REGION Network 8: MATERIAL ADDITION PROCESS SELECT
   RUNG wire#powerrail
      { S7_Templates := "SrcType := Int" } EQ_Contact(in1 := "MODE SELECTION DB"."MODE BUFF", in2 := 1)
      { S7_Templates := "SrcType := Int" } EQ_Contact(in1 := "MFG PROCESS_DB"."AUTO BUFF", in2 := 60)
      Coil( "AUTO ALARM DB"."MFG PROCESS"."MATERIAL ADDITION PROCESS SELECT" )
   END_RUNG
   // the same network as SCL:
   "AUTO ALARM DB"."MFG PROCESS"."MATERIAL ADDITION PROCESS SELECT" := ("MODE SELECTION DB"."MODE BUFF" = 1) AND ("MFG PROCESS_DB"."AUTO BUFF" = 60);
END_REGION

REGION Network 9: MATERIAL ADDITION MATERIAL ADDED TEXT
   RUNG wire#powerrail
      { S7_Templates := "SrcType := Int" } EQ_Contact(in1 := "MODE SELECTION DB"."MODE BUFF", in2 := 1)
      { S7_Templates := "SrcType := Int" } EQ_Contact(in1 := "MFG PROCESS_DB"."AUTO BUFF", in2 := 65)
      Coil( "AUTO ALARM DB"."MFG PROCESS"."MATERIAL ADDITION MATERIAL ADDED TEXT" )
   END_RUNG
   // the same network as SCL:
   "AUTO ALARM DB"."MFG PROCESS"."MATERIAL ADDITION MATERIAL ADDED TEXT" := ("MODE SELECTION DB"."MODE BUFF" = 1) AND ("MFG PROCESS_DB"."AUTO BUFF" = 65);
END_REGION

REGION Network 10: MATERIAL ADDITION DO YOU WANT TO ADD SORBITOL SELECT
   RUNG wire#powerrail
      { S7_Templates := "SrcType := Int" } EQ_Contact(in1 := "MODE SELECTION DB"."MODE BUFF", in2 := 1)
      { S7_Templates := "SrcType := Int" } EQ_Contact(in1 := "MFG PROCESS_DB"."AUTO BUFF", in2 := 75)
      Coil( "AUTO ALARM DB"."MFG PROCESS"."MATERIAL ADDITION DO YOU WANT TO ADD SORBITOL SELECT" )
   END_RUNG
   // the same network as SCL:
   "AUTO ALARM DB"."MFG PROCESS"."MATERIAL ADDITION DO YOU WANT TO ADD SORBITOL SELECT" := ("MODE SELECTION DB"."MODE BUFF" = 1) AND ("MFG PROCESS_DB"."AUTO BUFF" = 75);
END_REGION

REGION Network 11: MATERIAL ADDITION OF SORBITOL OVER
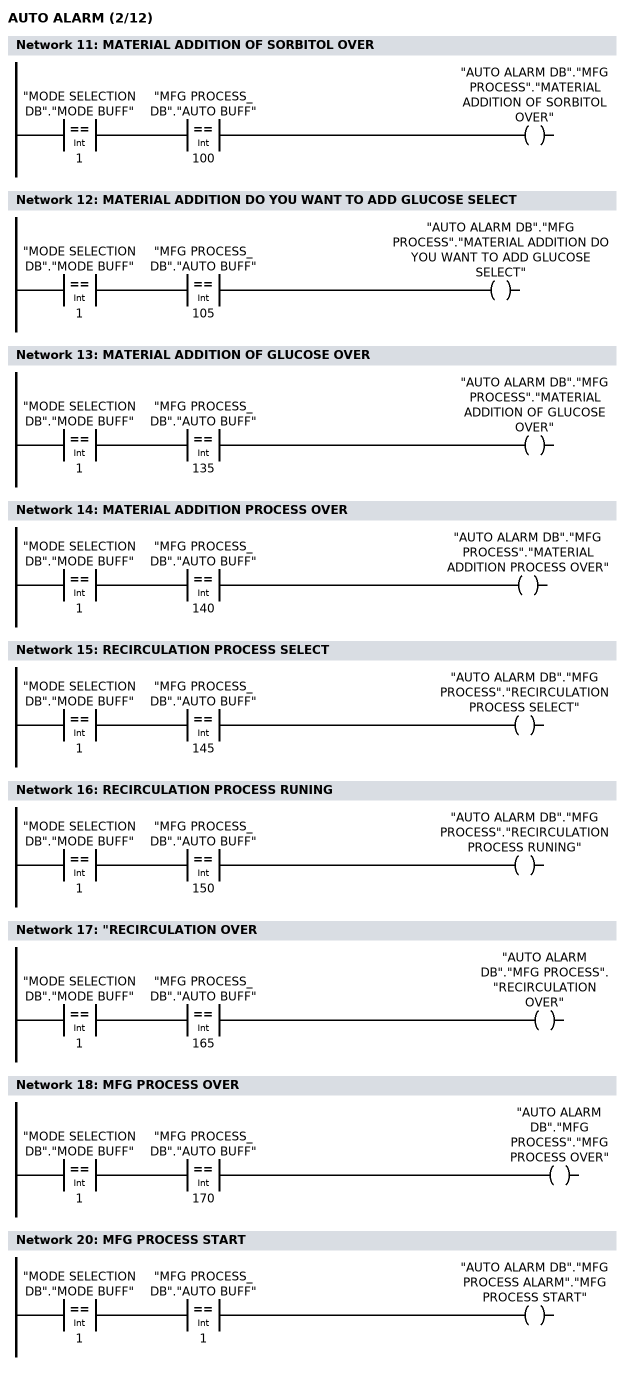
   RUNG wire#powerrail
      { S7_Templates := "SrcType := Int" } EQ_Contact(in1 := "MODE SELECTION DB"."MODE BUFF", in2 := 1)
      { S7_Templates := "SrcType := Int" } EQ_Contact(in1 := "MFG PROCESS_DB"."AUTO BUFF", in2 := 100)
      Coil( "AUTO ALARM DB"."MFG PROCESS"."MATERIAL ADDITION OF SORBITOL OVER" )
   END_RUNG
   // the same network as SCL:
   "AUTO ALARM DB"."MFG PROCESS"."MATERIAL ADDITION OF SORBITOL OVER" := ("MODE SELECTION DB"."MODE BUFF" = 1) AND ("MFG PROCESS_DB"."AUTO BUFF" = 100);
END_REGION

REGION Network 12: MATERIAL ADDITION DO YOU WANT TO ADD GLUCOSE SELECT
   RUNG wire#powerrail
      { S7_Templates := "SrcType := Int" } EQ_Contact(in1 := "MODE SELECTION DB"."MODE BUFF", in2 := 1)
      { S7_Templates := "SrcType := Int" } EQ_Contact(in1 := "MFG PROCESS_DB"."AUTO BUFF", in2 := 105)
      Coil( "AUTO ALARM DB"."MFG PROCESS"."MATERIAL ADDITION DO YOU WANT TO ADD GLUCOSE SELECT" )
   END_RUNG
   // the same network as SCL:
   "AUTO ALARM DB"."MFG PROCESS"."MATERIAL ADDITION DO YOU WANT TO ADD GLUCOSE SELECT" := ("MODE SELECTION DB"."MODE BUFF" = 1) AND ("MFG PROCESS_DB"."AUTO BUFF" = 105);
END_REGION

REGION Network 13: MATERIAL ADDITION OF GLUCOSE OVER
   RUNG wire#powerrail
      { S7_Templates := "SrcType := Int" } EQ_Contact(in1 := "MODE SELECTION DB"."MODE BUFF", in2 := 1)
      { S7_Templates := "SrcType := Int" } EQ_Contact(in1 := "MFG PROCESS_DB"."AUTO BUFF", in2 := 135)
      Coil( "AUTO ALARM DB"."MFG PROCESS"."MATERIAL ADDITION OF GLUCOSE OVER" )
   END_RUNG
   // the same network as SCL:
   "AUTO ALARM DB"."MFG PROCESS"."MATERIAL ADDITION OF GLUCOSE OVER" := ("MODE SELECTION DB"."MODE BUFF" = 1) AND ("MFG PROCESS_DB"."AUTO BUFF" = 135);
END_REGION

REGION Network 14: MATERIAL ADDITION PROCESS OVER
   RUNG wire#powerrail
      { S7_Templates := "SrcType := Int" } EQ_Contact(in1 := "MODE SELECTION DB"."MODE BUFF", in2 := 1)
      { S7_Templates := "SrcType := Int" } EQ_Contact(in1 := "MFG PROCESS_DB"."AUTO BUFF", in2 := 140)
      Coil( "AUTO ALARM DB"."MFG PROCESS"."MATERIAL ADDITION PROCESS OVER" )
   END_RUNG
   // the same network as SCL:
   "AUTO ALARM DB"."MFG PROCESS"."MATERIAL ADDITION PROCESS OVER" := ("MODE SELECTION DB"."MODE BUFF" = 1) AND ("MFG PROCESS_DB"."AUTO BUFF" = 140);
END_REGION

REGION Network 15: RECIRCULATION PROCESS SELECT
   RUNG wire#powerrail
      { S7_Templates := "SrcType := Int" } EQ_Contact(in1 := "MODE SELECTION DB"."MODE BUFF", in2 := 1)
      { S7_Templates := "SrcType := Int" } EQ_Contact(in1 := "MFG PROCESS_DB"."AUTO BUFF", in2 := 145)
      Coil( "AUTO ALARM DB"."MFG PROCESS"."RECIRCULATION PROCESS SELECT" )
   END_RUNG
   // the same network as SCL:
   "AUTO ALARM DB"."MFG PROCESS"."RECIRCULATION PROCESS SELECT" := ("MODE SELECTION DB"."MODE BUFF" = 1) AND ("MFG PROCESS_DB"."AUTO BUFF" = 145);
END_REGION

REGION Network 16: RECIRCULATION PROCESS RUNING
   RUNG wire#powerrail
      { S7_Templates := "SrcType := Int" } EQ_Contact(in1 := "MODE SELECTION DB"."MODE BUFF", in2 := 1)
      { S7_Templates := "SrcType := Int" } EQ_Contact(in1 := "MFG PROCESS_DB"."AUTO BUFF", in2 := 150)
      Coil( "AUTO ALARM DB"."MFG PROCESS"."RECIRCULATION PROCESS RUNING" )
   END_RUNG
   // the same network as SCL:
   "AUTO ALARM DB"."MFG PROCESS"."RECIRCULATION PROCESS RUNING" := ("MODE SELECTION DB"."MODE BUFF" = 1) AND ("MFG PROCESS_DB"."AUTO BUFF" = 150);
END_REGION

REGION Network 17: "RECIRCULATION OVER
   RUNG wire#powerrail
      { S7_Templates := "SrcType := Int" } EQ_Contact(in1 := "MODE SELECTION DB"."MODE BUFF", in2 := 1)
      { S7_Templates := "SrcType := Int" } EQ_Contact(in1 := "MFG PROCESS_DB"."AUTO BUFF", in2 := 165)
      Coil( "AUTO ALARM DB"."MFG PROCESS"."RECIRCULATION OVER" )
   END_RUNG
   // the same network as SCL:
   "AUTO ALARM DB"."MFG PROCESS"."RECIRCULATION OVER" := ("MODE SELECTION DB"."MODE BUFF" = 1) AND ("MFG PROCESS_DB"."AUTO BUFF" = 165);
END_REGION

REGION Network 18: MFG PROCESS OVER
   RUNG wire#powerrail
      { S7_Templates := "SrcType := Int" } EQ_Contact(in1 := "MODE SELECTION DB"."MODE BUFF", in2 := 1)
      { S7_Templates := "SrcType := Int" } EQ_Contact(in1 := "MFG PROCESS_DB"."AUTO BUFF", in2 := 170)
      Coil( "AUTO ALARM DB"."MFG PROCESS"."MFG PROCESS OVER" )
   END_RUNG
   // the same network as SCL:
   "AUTO ALARM DB"."MFG PROCESS"."MFG PROCESS OVER" := ("MODE SELECTION DB"."MODE BUFF" = 1) AND ("MFG PROCESS_DB"."AUTO BUFF" = 170);
END_REGION

REGION Network 19: ///////////////////////////////MFG ALARM /////////////////////////////////////
END_REGION

REGION Network 20: MFG PROCESS START
   RUNG wire#powerrail
      { S7_Templates := "SrcType := Int" } EQ_Contact(in1 := "MODE SELECTION DB"."MODE BUFF", in2 := 1)
      { S7_Templates := "SrcType := Int" } EQ_Contact(in1 := "MFG PROCESS_DB"."AUTO BUFF", in2 := 1)
      Coil( "AUTO ALARM DB"."MFG PROCESS ALARM"."MFG PROCESS START" )
   END_RUNG
   // the same network as SCL:
   "AUTO ALARM DB"."MFG PROCESS ALARM"."MFG PROCESS START" := ("MODE SELECTION DB"."MODE BUFF" = 1) AND ("MFG PROCESS_DB"."AUTO BUFF" = 1);
END_REGION

REGION Network 21: PURIFIED WATER PROCESS START
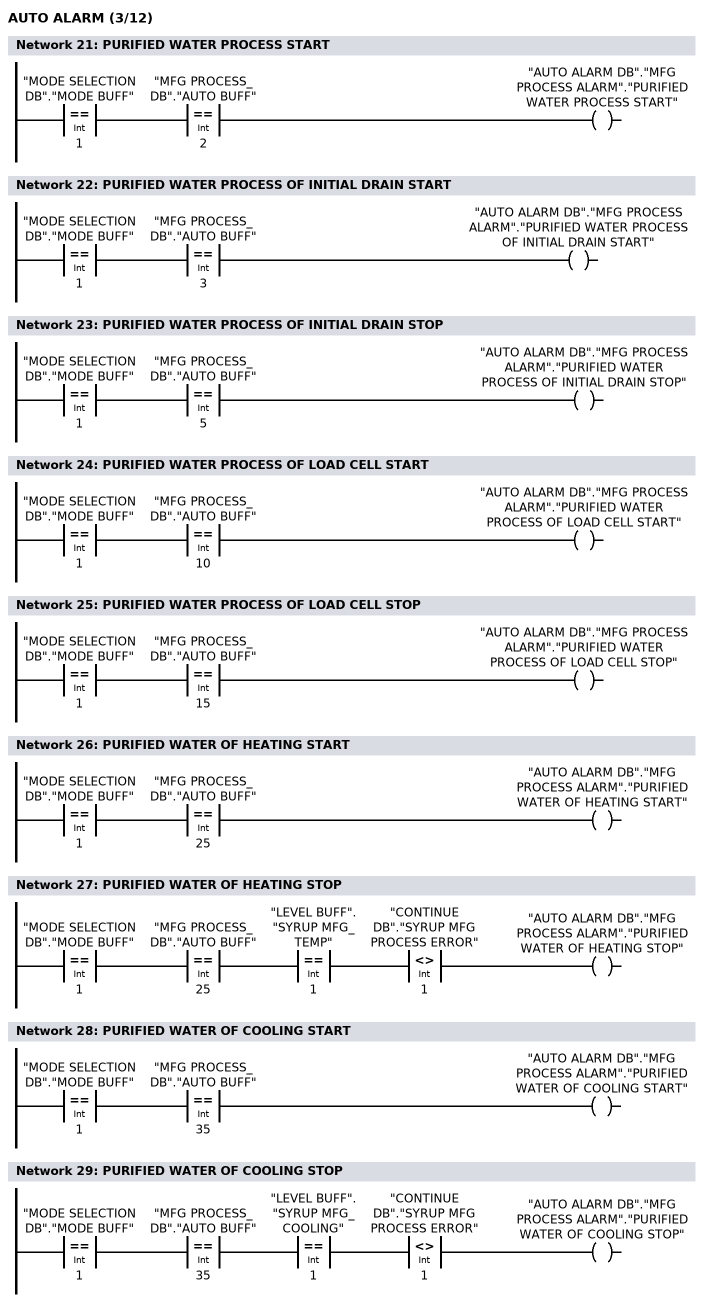
   RUNG wire#powerrail
      { S7_Templates := "SrcType := Int" } EQ_Contact(in1 := "MODE SELECTION DB"."MODE BUFF", in2 := 1)
      { S7_Templates := "SrcType := Int" } EQ_Contact(in1 := "MFG PROCESS_DB"."AUTO BUFF", in2 := 2)
      Coil( "AUTO ALARM DB"."MFG PROCESS ALARM"."PURIFIED WATER PROCESS START" )
   END_RUNG
   // the same network as SCL:
   "AUTO ALARM DB"."MFG PROCESS ALARM"."PURIFIED WATER PROCESS START" := ("MODE SELECTION DB"."MODE BUFF" = 1) AND ("MFG PROCESS_DB"."AUTO BUFF" = 2);
END_REGION

REGION Network 22: PURIFIED WATER PROCESS OF INITIAL DRAIN START
   RUNG wire#powerrail
      { S7_Templates := "SrcType := Int" } EQ_Contact(in1 := "MODE SELECTION DB"."MODE BUFF", in2 := 1)
      { S7_Templates := "SrcType := Int" } EQ_Contact(in1 := "MFG PROCESS_DB"."AUTO BUFF", in2 := 3)
      Coil( "AUTO ALARM DB"."MFG PROCESS ALARM"."PURIFIED WATER PROCESS OF INITIAL DRAIN START" )
   END_RUNG
   // the same network as SCL:
   "AUTO ALARM DB"."MFG PROCESS ALARM"."PURIFIED WATER PROCESS OF INITIAL DRAIN START" := ("MODE SELECTION DB"."MODE BUFF" = 1) AND ("MFG PROCESS_DB"."AUTO BUFF" = 3);
END_REGION

REGION Network 23: PURIFIED WATER PROCESS OF INITIAL DRAIN STOP
   RUNG wire#powerrail
      { S7_Templates := "SrcType := Int" } EQ_Contact(in1 := "MODE SELECTION DB"."MODE BUFF", in2 := 1)
      { S7_Templates := "SrcType := Int" } EQ_Contact(in1 := "MFG PROCESS_DB"."AUTO BUFF", in2 := 5)
      Coil( "AUTO ALARM DB"."MFG PROCESS ALARM"."PURIFIED WATER PROCESS OF INITIAL DRAIN STOP" )
   END_RUNG
   // the same network as SCL:
   "AUTO ALARM DB"."MFG PROCESS ALARM"."PURIFIED WATER PROCESS OF INITIAL DRAIN STOP" := ("MODE SELECTION DB"."MODE BUFF" = 1) AND ("MFG PROCESS_DB"."AUTO BUFF" = 5);
END_REGION

REGION Network 24: PURIFIED WATER PROCESS OF LOAD CELL START
   RUNG wire#powerrail
      { S7_Templates := "SrcType := Int" } EQ_Contact(in1 := "MODE SELECTION DB"."MODE BUFF", in2 := 1)
      { S7_Templates := "SrcType := Int" } EQ_Contact(in1 := "MFG PROCESS_DB"."AUTO BUFF", in2 := 10)
      Coil( "AUTO ALARM DB"."MFG PROCESS ALARM"."PURIFIED WATER PROCESS OF LOAD CELL START" )
   END_RUNG
   // the same network as SCL:
   "AUTO ALARM DB"."MFG PROCESS ALARM"."PURIFIED WATER PROCESS OF LOAD CELL START" := ("MODE SELECTION DB"."MODE BUFF" = 1) AND ("MFG PROCESS_DB"."AUTO BUFF" = 10);
END_REGION

REGION Network 25: PURIFIED WATER PROCESS OF LOAD CELL STOP
   RUNG wire#powerrail
      { S7_Templates := "SrcType := Int" } EQ_Contact(in1 := "MODE SELECTION DB"."MODE BUFF", in2 := 1)
      { S7_Templates := "SrcType := Int" } EQ_Contact(in1 := "MFG PROCESS_DB"."AUTO BUFF", in2 := 15)
      Coil( "AUTO ALARM DB"."MFG PROCESS ALARM"."PURIFIED WATER PROCESS OF LOAD CELL STOP" )
   END_RUNG
   // the same network as SCL:
   "AUTO ALARM DB"."MFG PROCESS ALARM"."PURIFIED WATER PROCESS OF LOAD CELL STOP" := ("MODE SELECTION DB"."MODE BUFF" = 1) AND ("MFG PROCESS_DB"."AUTO BUFF" = 15);
END_REGION

REGION Network 26: PURIFIED WATER OF HEATING START
   RUNG wire#powerrail
      { S7_Templates := "SrcType := Int" } EQ_Contact(in1 := "MODE SELECTION DB"."MODE BUFF", in2 := 1)
      { S7_Templates := "SrcType := Int" } EQ_Contact(in1 := "MFG PROCESS_DB"."AUTO BUFF", in2 := 25)
      Coil( "AUTO ALARM DB"."MFG PROCESS ALARM"."PURIFIED WATER OF HEATING START" )
   END_RUNG
   // the same network as SCL:
   "AUTO ALARM DB"."MFG PROCESS ALARM"."PURIFIED WATER OF HEATING START" := ("MODE SELECTION DB"."MODE BUFF" = 1) AND ("MFG PROCESS_DB"."AUTO BUFF" = 25);
END_REGION

REGION Network 27: PURIFIED WATER OF HEATING STOP
   RUNG wire#powerrail
      { S7_Templates := "SrcType := Int" } EQ_Contact(in1 := "MODE SELECTION DB"."MODE BUFF", in2 := 1)
      { S7_Templates := "SrcType := Int" } EQ_Contact(in1 := "MFG PROCESS_DB"."AUTO BUFF", in2 := 25)
      { S7_Templates := "SrcType := Int" } EQ_Contact(in1 := "LEVEL BUFF"."SYRUP MFG_TEMP", in2 := 1)
      { S7_Templates := "SrcType := Int" } NE_Contact(in1 := "CONTINUE DB"."SYRUP MFG PROCESS ERROR", in2 := 1)
      Coil( "AUTO ALARM DB"."MFG PROCESS ALARM"."PURIFIED WATER OF HEATING STOP" )
   END_RUNG
   // the same network as SCL:
   "AUTO ALARM DB"."MFG PROCESS ALARM"."PURIFIED WATER OF HEATING STOP" := ("MODE SELECTION DB"."MODE BUFF" = 1) AND ("MFG PROCESS_DB"."AUTO BUFF" = 25) AND ("LEVEL BUFF"."SYRUP MFG_TEMP" = 1) AND ("CONTINUE DB"."SYRUP MFG PROCESS ERROR" <> 1);
END_REGION

REGION Network 28: PURIFIED WATER OF COOLING START
   RUNG wire#powerrail
      { S7_Templates := "SrcType := Int" } EQ_Contact(in1 := "MODE SELECTION DB"."MODE BUFF", in2 := 1)
      { S7_Templates := "SrcType := Int" } EQ_Contact(in1 := "MFG PROCESS_DB"."AUTO BUFF", in2 := 35)
      Coil( "AUTO ALARM DB"."MFG PROCESS ALARM"."PURIFIED WATER OF COOLING START" )
   END_RUNG
   // the same network as SCL:
   "AUTO ALARM DB"."MFG PROCESS ALARM"."PURIFIED WATER OF COOLING START" := ("MODE SELECTION DB"."MODE BUFF" = 1) AND ("MFG PROCESS_DB"."AUTO BUFF" = 35);
END_REGION

REGION Network 29: PURIFIED WATER OF COOLING STOP
   RUNG wire#powerrail
      { S7_Templates := "SrcType := Int" } EQ_Contact(in1 := "MODE SELECTION DB"."MODE BUFF", in2 := 1)
      { S7_Templates := "SrcType := Int" } EQ_Contact(in1 := "MFG PROCESS_DB"."AUTO BUFF", in2 := 35)
      { S7_Templates := "SrcType := Int" } EQ_Contact(in1 := "LEVEL BUFF"."SYRUP MFG_COOLING", in2 := 1)
      { S7_Templates := "SrcType := Int" } NE_Contact(in1 := "CONTINUE DB"."SYRUP MFG PROCESS ERROR", in2 := 1)
      Coil( "AUTO ALARM DB"."MFG PROCESS ALARM"."PURIFIED WATER OF COOLING STOP" )
   END_RUNG
   // the same network as SCL:
   "AUTO ALARM DB"."MFG PROCESS ALARM"."PURIFIED WATER OF COOLING STOP" := ("MODE SELECTION DB"."MODE BUFF" = 1) AND ("MFG PROCESS_DB"."AUTO BUFF" = 35) AND ("LEVEL BUFF"."SYRUP MFG_COOLING" = 1) AND ("CONTINUE DB"."SYRUP MFG PROCESS ERROR" <> 1);
END_REGION

REGION Network 30: PURIFIED WATER PROCESS OF JACKET DRAIN START
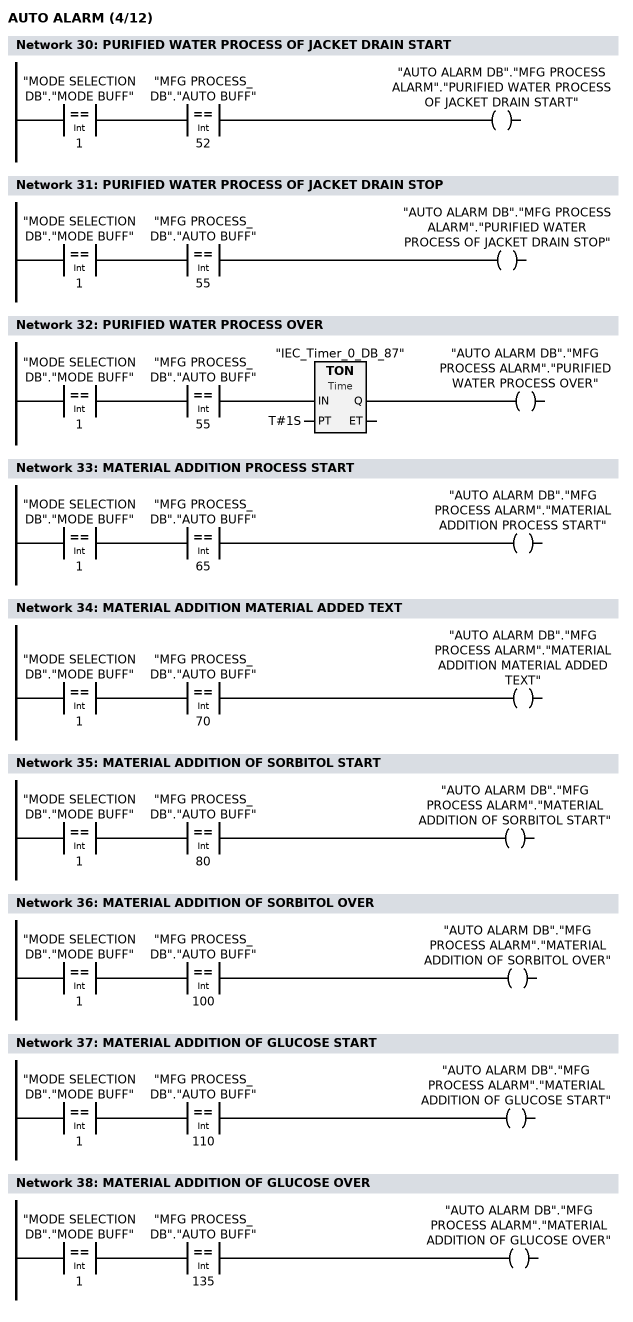
   RUNG wire#powerrail
      { S7_Templates := "SrcType := Int" } EQ_Contact(in1 := "MODE SELECTION DB"."MODE BUFF", in2 := 1)
      { S7_Templates := "SrcType := Int" } EQ_Contact(in1 := "MFG PROCESS_DB"."AUTO BUFF", in2 := 52)
      Coil( "AUTO ALARM DB"."MFG PROCESS ALARM"."PURIFIED WATER PROCESS OF JACKET DRAIN START" )
   END_RUNG
   // the same network as SCL:
   "AUTO ALARM DB"."MFG PROCESS ALARM"."PURIFIED WATER PROCESS OF JACKET DRAIN START" := ("MODE SELECTION DB"."MODE BUFF" = 1) AND ("MFG PROCESS_DB"."AUTO BUFF" = 52);
END_REGION

REGION Network 31: PURIFIED WATER PROCESS OF JACKET DRAIN STOP
   RUNG wire#powerrail
      { S7_Templates := "SrcType := Int" } EQ_Contact(in1 := "MODE SELECTION DB"."MODE BUFF", in2 := 1)
      { S7_Templates := "SrcType := Int" } EQ_Contact(in1 := "MFG PROCESS_DB"."AUTO BUFF", in2 := 55)
      Coil( "AUTO ALARM DB"."MFG PROCESS ALARM"."PURIFIED WATER PROCESS OF JACKET DRAIN STOP" )
   END_RUNG
   // the same network as SCL:
   "AUTO ALARM DB"."MFG PROCESS ALARM"."PURIFIED WATER PROCESS OF JACKET DRAIN STOP" := ("MODE SELECTION DB"."MODE BUFF" = 1) AND ("MFG PROCESS_DB"."AUTO BUFF" = 55);
END_REGION

REGION Network 32: PURIFIED WATER PROCESS OVER
   RUNG wire#powerrail
      { S7_Templates := "SrcType := Int" } EQ_Contact(in1 := "MODE SELECTION DB"."MODE BUFF", in2 := 1)
      { S7_Templates := "SrcType := Int" } EQ_Contact(in1 := "MFG PROCESS_DB"."AUTO BUFF", in2 := 55)
      { S7_Templates := "time_type := Time" } "IEC_Timer_0_DB_87".TON(pt := T#1S, et =>)
      Coil( "AUTO ALARM DB"."MFG PROCESS ALARM"."PURIFIED WATER PROCESS OVER" )
   END_RUNG
   // the same network as SCL:
   "IEC_Timer_0_DB_87".TON(IN := ("MODE SELECTION DB"."MODE BUFF" = 1) AND ("MFG PROCESS_DB"."AUTO BUFF" = 55),
                           PT := T#1S);
   "AUTO ALARM DB"."MFG PROCESS ALARM"."PURIFIED WATER PROCESS OVER" := "IEC_Timer_0_DB_87".Q;
END_REGION

REGION Network 33: MATERIAL ADDITION PROCESS START
   RUNG wire#powerrail
      { S7_Templates := "SrcType := Int" } EQ_Contact(in1 := "MODE SELECTION DB"."MODE BUFF", in2 := 1)
      { S7_Templates := "SrcType := Int" } EQ_Contact(in1 := "MFG PROCESS_DB"."AUTO BUFF", in2 := 65)
      Coil( "AUTO ALARM DB"."MFG PROCESS ALARM"."MATERIAL ADDITION PROCESS START" )
   END_RUNG
   // the same network as SCL:
   "AUTO ALARM DB"."MFG PROCESS ALARM"."MATERIAL ADDITION PROCESS START" := ("MODE SELECTION DB"."MODE BUFF" = 1) AND ("MFG PROCESS_DB"."AUTO BUFF" = 65);
END_REGION

REGION Network 34: MATERIAL ADDITION MATERIAL ADDED TEXT
   RUNG wire#powerrail
      { S7_Templates := "SrcType := Int" } EQ_Contact(in1 := "MODE SELECTION DB"."MODE BUFF", in2 := 1)
      { S7_Templates := "SrcType := Int" } EQ_Contact(in1 := "MFG PROCESS_DB"."AUTO BUFF", in2 := 70)
      Coil( "AUTO ALARM DB"."MFG PROCESS ALARM"."MATERIAL ADDITION MATERIAL ADDED TEXT" )
   END_RUNG
   // the same network as SCL:
   "AUTO ALARM DB"."MFG PROCESS ALARM"."MATERIAL ADDITION MATERIAL ADDED TEXT" := ("MODE SELECTION DB"."MODE BUFF" = 1) AND ("MFG PROCESS_DB"."AUTO BUFF" = 70);
END_REGION

REGION Network 35: MATERIAL ADDITION OF SORBITOL START
   RUNG wire#powerrail
      { S7_Templates := "SrcType := Int" } EQ_Contact(in1 := "MODE SELECTION DB"."MODE BUFF", in2 := 1)
      { S7_Templates := "SrcType := Int" } EQ_Contact(in1 := "MFG PROCESS_DB"."AUTO BUFF", in2 := 80)
      Coil( "AUTO ALARM DB"."MFG PROCESS ALARM"."MATERIAL ADDITION OF SORBITOL START" )
   END_RUNG
   // the same network as SCL:
   "AUTO ALARM DB"."MFG PROCESS ALARM"."MATERIAL ADDITION OF SORBITOL START" := ("MODE SELECTION DB"."MODE BUFF" = 1) AND ("MFG PROCESS_DB"."AUTO BUFF" = 80);
END_REGION

REGION Network 36: MATERIAL ADDITION OF SORBITOL OVER
   RUNG wire#powerrail
      { S7_Templates := "SrcType := Int" } EQ_Contact(in1 := "MODE SELECTION DB"."MODE BUFF", in2 := 1)
      { S7_Templates := "SrcType := Int" } EQ_Contact(in1 := "MFG PROCESS_DB"."AUTO BUFF", in2 := 100)
      Coil( "AUTO ALARM DB"."MFG PROCESS ALARM"."MATERIAL ADDITION OF SORBITOL OVER" )
   END_RUNG
   // the same network as SCL:
   "AUTO ALARM DB"."MFG PROCESS ALARM"."MATERIAL ADDITION OF SORBITOL OVER" := ("MODE SELECTION DB"."MODE BUFF" = 1) AND ("MFG PROCESS_DB"."AUTO BUFF" = 100);
END_REGION

REGION Network 37: MATERIAL ADDITION OF GLUCOSE START
   RUNG wire#powerrail
      { S7_Templates := "SrcType := Int" } EQ_Contact(in1 := "MODE SELECTION DB"."MODE BUFF", in2 := 1)
      { S7_Templates := "SrcType := Int" } EQ_Contact(in1 := "MFG PROCESS_DB"."AUTO BUFF", in2 := 110)
      Coil( "AUTO ALARM DB"."MFG PROCESS ALARM"."MATERIAL ADDITION OF GLUCOSE START" )
   END_RUNG
   // the same network as SCL:
   "AUTO ALARM DB"."MFG PROCESS ALARM"."MATERIAL ADDITION OF GLUCOSE START" := ("MODE SELECTION DB"."MODE BUFF" = 1) AND ("MFG PROCESS_DB"."AUTO BUFF" = 110);
END_REGION

REGION Network 38: MATERIAL ADDITION OF GLUCOSE OVER
   RUNG wire#powerrail
      { S7_Templates := "SrcType := Int" } EQ_Contact(in1 := "MODE SELECTION DB"."MODE BUFF", in2 := 1)
      { S7_Templates := "SrcType := Int" } EQ_Contact(in1 := "MFG PROCESS_DB"."AUTO BUFF", in2 := 135)
      Coil( "AUTO ALARM DB"."MFG PROCESS ALARM"."MATERIAL ADDITION OF GLUCOSE OVER" )
   END_RUNG
   // the same network as SCL:
   "AUTO ALARM DB"."MFG PROCESS ALARM"."MATERIAL ADDITION OF GLUCOSE OVER" := ("MODE SELECTION DB"."MODE BUFF" = 1) AND ("MFG PROCESS_DB"."AUTO BUFF" = 135);
END_REGION

REGION Network 39: MATERIAL ADDITION PROCESS OVER
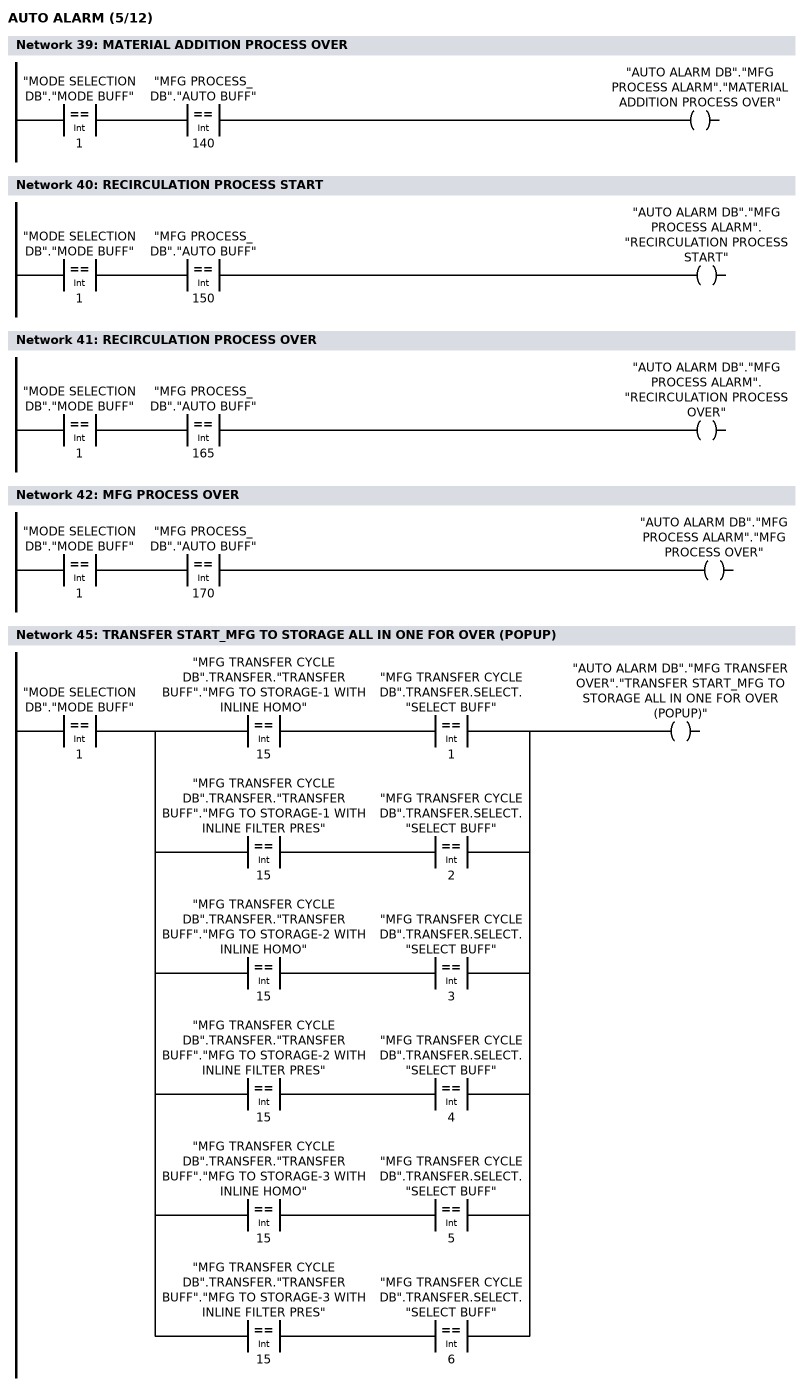
   RUNG wire#powerrail
      { S7_Templates := "SrcType := Int" } EQ_Contact(in1 := "MODE SELECTION DB"."MODE BUFF", in2 := 1)
      { S7_Templates := "SrcType := Int" } EQ_Contact(in1 := "MFG PROCESS_DB"."AUTO BUFF", in2 := 140)
      Coil( "AUTO ALARM DB"."MFG PROCESS ALARM"."MATERIAL ADDITION PROCESS OVER" )
   END_RUNG
   // the same network as SCL:
   "AUTO ALARM DB"."MFG PROCESS ALARM"."MATERIAL ADDITION PROCESS OVER" := ("MODE SELECTION DB"."MODE BUFF" = 1) AND ("MFG PROCESS_DB"."AUTO BUFF" = 140);
END_REGION

REGION Network 40: RECIRCULATION PROCESS START
   RUNG wire#powerrail
      { S7_Templates := "SrcType := Int" } EQ_Contact(in1 := "MODE SELECTION DB"."MODE BUFF", in2 := 1)
      { S7_Templates := "SrcType := Int" } EQ_Contact(in1 := "MFG PROCESS_DB"."AUTO BUFF", in2 := 150)
      Coil( "AUTO ALARM DB"."MFG PROCESS ALARM"."RECIRCULATION PROCESS START" )
   END_RUNG
   // the same network as SCL:
   "AUTO ALARM DB"."MFG PROCESS ALARM"."RECIRCULATION PROCESS START" := ("MODE SELECTION DB"."MODE BUFF" = 1) AND ("MFG PROCESS_DB"."AUTO BUFF" = 150);
END_REGION

REGION Network 41: RECIRCULATION PROCESS OVER
   RUNG wire#powerrail
      { S7_Templates := "SrcType := Int" } EQ_Contact(in1 := "MODE SELECTION DB"."MODE BUFF", in2 := 1)
      { S7_Templates := "SrcType := Int" } EQ_Contact(in1 := "MFG PROCESS_DB"."AUTO BUFF", in2 := 165)
      Coil( "AUTO ALARM DB"."MFG PROCESS ALARM"."RECIRCULATION PROCESS OVER" )
   END_RUNG
   // the same network as SCL:
   "AUTO ALARM DB"."MFG PROCESS ALARM"."RECIRCULATION PROCESS OVER" := ("MODE SELECTION DB"."MODE BUFF" = 1) AND ("MFG PROCESS_DB"."AUTO BUFF" = 165);
END_REGION

REGION Network 42: MFG PROCESS OVER
   RUNG wire#powerrail
      { S7_Templates := "SrcType := Int" } EQ_Contact(in1 := "MODE SELECTION DB"."MODE BUFF", in2 := 1)
      { S7_Templates := "SrcType := Int" } EQ_Contact(in1 := "MFG PROCESS_DB"."AUTO BUFF", in2 := 170)
      Coil( "AUTO ALARM DB"."MFG PROCESS ALARM"."MFG PROCESS OVER" )
   END_RUNG
   // the same network as SCL:
   "AUTO ALARM DB"."MFG PROCESS ALARM"."MFG PROCESS OVER" := ("MODE SELECTION DB"."MODE BUFF" = 1) AND ("MFG PROCESS_DB"."AUTO BUFF" = 170);
END_REGION

REGION Network 45: TRANSFER START_MFG TO STORAGE ALL IN ONE FOR OVER (POPUP)
   RUNG wire#powerrail
      { S7_Templates := "SrcType := Int" } EQ_Contact(in1 := "MODE SELECTION DB"."MODE BUFF", in2 := 1)
      wire#w1
      { S7_Templates := "SrcType := Int" } EQ_Contact(in1 := "MFG TRANSFER CYCLE DB".TRANSFER."TRANSFER BUFF"."MFG TO STORAGE-1 WITH INLINE HOMO", in2 := 15)
      { S7_Templates := "SrcType := Int" } EQ_Contact(in1 := "MFG TRANSFER CYCLE DB".TRANSFER.SELECT."SELECT BUFF", in2 := 1)
      wire#w2
      Coil( "AUTO ALARM DB"."MFG TRANSFER OVER"."TRANSFER START_MFG TO STORAGE ALL IN ONE FOR OVER (POPUP)" )
   END_RUNG
   RUNG wire#w1
      { S7_Templates := "SrcType := Int" } EQ_Contact(in1 := "MFG TRANSFER CYCLE DB".TRANSFER."TRANSFER BUFF"."MFG TO STORAGE-1 WITH INLINE FILTER PRES", in2 := 15)
      { S7_Templates := "SrcType := Int" } EQ_Contact(in1 := "MFG TRANSFER CYCLE DB".TRANSFER.SELECT."SELECT BUFF", in2 := 2)
   END_RUNG wire#w2
   RUNG wire#w1
      { S7_Templates := "SrcType := Int" } EQ_Contact(in1 := "MFG TRANSFER CYCLE DB".TRANSFER."TRANSFER BUFF"."MFG TO STORAGE-2 WITH INLINE HOMO", in2 := 15)
      { S7_Templates := "SrcType := Int" } EQ_Contact(in1 := "MFG TRANSFER CYCLE DB".TRANSFER.SELECT."SELECT BUFF", in2 := 3)
   END_RUNG wire#w2
   RUNG wire#w1
      { S7_Templates := "SrcType := Int" } EQ_Contact(in1 := "MFG TRANSFER CYCLE DB".TRANSFER."TRANSFER BUFF"."MFG TO STORAGE-2 WITH INLINE FILTER PRES", in2 := 15)
      { S7_Templates := "SrcType := Int" } EQ_Contact(in1 := "MFG TRANSFER CYCLE DB".TRANSFER.SELECT."SELECT BUFF", in2 := 4)
   END_RUNG wire#w2
   RUNG wire#w1
      { S7_Templates := "SrcType := Int" } EQ_Contact(in1 := "MFG TRANSFER CYCLE DB".TRANSFER."TRANSFER BUFF"."MFG TO STORAGE-3 WITH INLINE HOMO", in2 := 15)
      { S7_Templates := "SrcType := Int" } EQ_Contact(in1 := "MFG TRANSFER CYCLE DB".TRANSFER.SELECT."SELECT BUFF", in2 := 5)
   END_RUNG wire#w2
   RUNG wire#w1
      { S7_Templates := "SrcType := Int" } EQ_Contact(in1 := "MFG TRANSFER CYCLE DB".TRANSFER."TRANSFER BUFF"."MFG TO STORAGE-3 WITH INLINE FILTER PRES", in2 := 15)
      { S7_Templates := "SrcType := Int" } EQ_Contact(in1 := "MFG TRANSFER CYCLE DB".TRANSFER.SELECT."SELECT BUFF", in2 := 6)
   END_RUNG wire#w2
   // the same network as SCL:
   "AUTO ALARM DB"."MFG TRANSFER OVER"."TRANSFER START_MFG TO STORAGE ALL IN ONE FOR OVER (POPUP)" := ("MODE SELECTION DB"."MODE BUFF" = 1) AND ((("MFG TRANSFER CYCLE DB".TRANSFER."TRANSFER BUFF"."MFG TO STORAGE-1 WITH INLINE HOMO" = 15) AND ("MFG TRANSFER CYCLE DB".TRANSFER.SELECT."SELECT BUFF" = 1)) OR (("MFG TRANSFER CYCLE DB".TRANSFER."TRANSFER BUFF"."MFG TO STORAGE-1 WITH INLINE FILTER PRES" = 15) AND ("MFG TRANSFER CYCLE DB".TRANSFER.SELECT."SELECT BUFF" = 2)) OR (("MFG TRANSFER CYCLE DB".TRANSFER."TRANSFER BUFF"."MFG TO STORAGE-2 WITH INLINE HOMO" = 15) AND ("MFG TRANSFER CYCLE DB".TRANSFER.SELECT."SELECT BUFF" = 3)) OR (("MFG TRANSFER CYCLE DB".TRANSFER."TRANSFER BUFF"."MFG TO STORAGE-2 WITH INLINE FILTER PRES" = 15) AND ("MFG TRANSFER CYCLE DB".TRANSFER.SELECT."SELECT BUFF" = 4)) OR (("MFG TRANSFER CYCLE DB".TRANSFER."TRANSFER BUFF"."MFG TO STORAGE-3 WITH INLINE HOMO" = 15) AND ("MFG TRANSFER CYCLE DB".TRANSFER.SELECT."SELECT BUFF" = 5)) OR (("MFG TRANSFER CYCLE DB".TRANSFER."TRANSFER BUFF"."MFG TO STORAGE-3 WITH INLINE FILTER PRES" = 15) AND ("MFG TRANSFER CYCLE DB".TRANSFER.SELECT."SELECT BUFF" = 6)));
END_REGION

REGION Network 46: TRANSFER START_MFG TO STORAGE-1 WITH INLINE HOMO
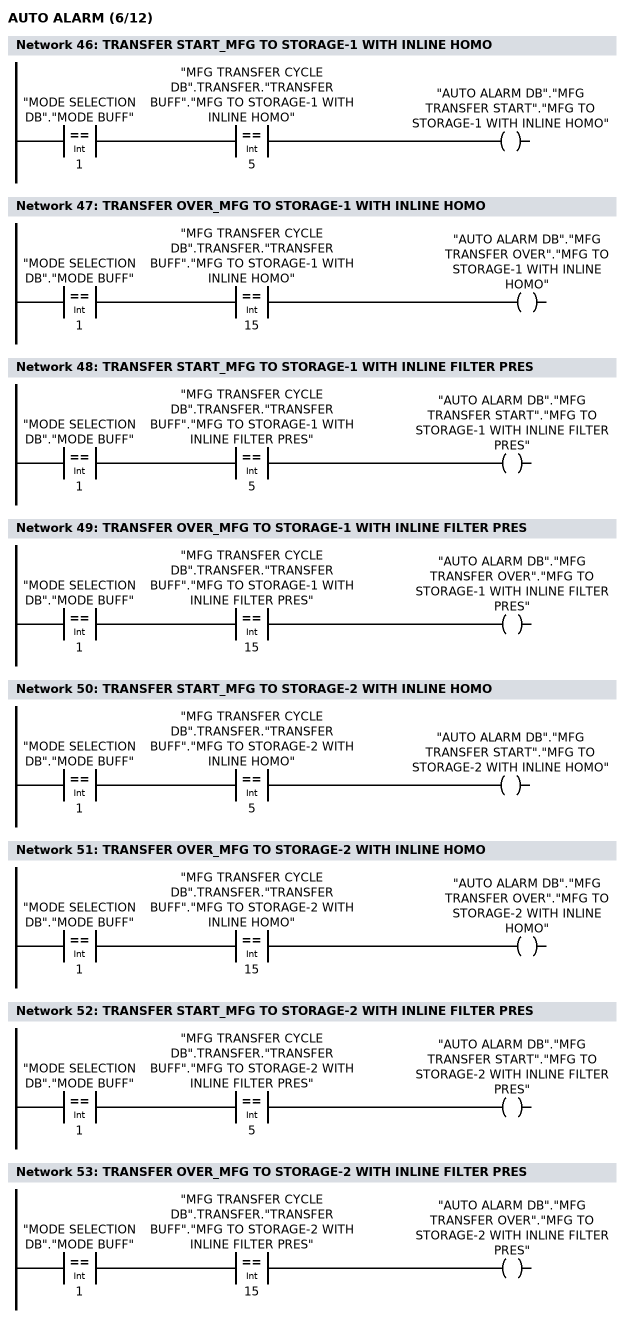
   RUNG wire#powerrail
      { S7_Templates := "SrcType := Int" } EQ_Contact(in1 := "MODE SELECTION DB"."MODE BUFF", in2 := 1)
      { S7_Templates := "SrcType := Int" } EQ_Contact(in1 := "MFG TRANSFER CYCLE DB".TRANSFER."TRANSFER BUFF"."MFG TO STORAGE-1 WITH INLINE HOMO", in2 := 5)
      Coil( "AUTO ALARM DB"."MFG TRANSFER START"."MFG TO STORAGE-1 WITH INLINE HOMO" )
   END_RUNG
   // the same network as SCL:
   "AUTO ALARM DB"."MFG TRANSFER START"."MFG TO STORAGE-1 WITH INLINE HOMO" := ("MODE SELECTION DB"."MODE BUFF" = 1) AND ("MFG TRANSFER CYCLE DB".TRANSFER."TRANSFER BUFF"."MFG TO STORAGE-1 WITH INLINE HOMO" = 5);
END_REGION

REGION Network 47: TRANSFER OVER_MFG TO STORAGE-1 WITH INLINE HOMO
   RUNG wire#powerrail
      { S7_Templates := "SrcType := Int" } EQ_Contact(in1 := "MODE SELECTION DB"."MODE BUFF", in2 := 1)
      { S7_Templates := "SrcType := Int" } EQ_Contact(in1 := "MFG TRANSFER CYCLE DB".TRANSFER."TRANSFER BUFF"."MFG TO STORAGE-1 WITH INLINE HOMO", in2 := 15)
      Coil( "AUTO ALARM DB"."MFG TRANSFER OVER"."MFG TO STORAGE-1 WITH INLINE HOMO" )
   END_RUNG
   // the same network as SCL:
   "AUTO ALARM DB"."MFG TRANSFER OVER"."MFG TO STORAGE-1 WITH INLINE HOMO" := ("MODE SELECTION DB"."MODE BUFF" = 1) AND ("MFG TRANSFER CYCLE DB".TRANSFER."TRANSFER BUFF"."MFG TO STORAGE-1 WITH INLINE HOMO" = 15);
END_REGION

REGION Network 48: TRANSFER START_MFG TO STORAGE-1 WITH INLINE FILTER PRES
   RUNG wire#powerrail
      { S7_Templates := "SrcType := Int" } EQ_Contact(in1 := "MODE SELECTION DB"."MODE BUFF", in2 := 1)
      { S7_Templates := "SrcType := Int" } EQ_Contact(in1 := "MFG TRANSFER CYCLE DB".TRANSFER."TRANSFER BUFF"."MFG TO STORAGE-1 WITH INLINE FILTER PRES", in2 := 5)
      Coil( "AUTO ALARM DB"."MFG TRANSFER START"."MFG TO STORAGE-1 WITH INLINE FILTER PRES" )
   END_RUNG
   // the same network as SCL:
   "AUTO ALARM DB"."MFG TRANSFER START"."MFG TO STORAGE-1 WITH INLINE FILTER PRES" := ("MODE SELECTION DB"."MODE BUFF" = 1) AND ("MFG TRANSFER CYCLE DB".TRANSFER."TRANSFER BUFF"."MFG TO STORAGE-1 WITH INLINE FILTER PRES" = 5);
END_REGION

REGION Network 49: TRANSFER OVER_MFG TO STORAGE-1 WITH INLINE FILTER PRES
   RUNG wire#powerrail
      { S7_Templates := "SrcType := Int" } EQ_Contact(in1 := "MODE SELECTION DB"."MODE BUFF", in2 := 1)
      { S7_Templates := "SrcType := Int" } EQ_Contact(in1 := "MFG TRANSFER CYCLE DB".TRANSFER."TRANSFER BUFF"."MFG TO STORAGE-1 WITH INLINE FILTER PRES", in2 := 15)
      Coil( "AUTO ALARM DB"."MFG TRANSFER OVER"."MFG TO STORAGE-1 WITH INLINE FILTER PRES" )
   END_RUNG
   // the same network as SCL:
   "AUTO ALARM DB"."MFG TRANSFER OVER"."MFG TO STORAGE-1 WITH INLINE FILTER PRES" := ("MODE SELECTION DB"."MODE BUFF" = 1) AND ("MFG TRANSFER CYCLE DB".TRANSFER."TRANSFER BUFF"."MFG TO STORAGE-1 WITH INLINE FILTER PRES" = 15);
END_REGION

REGION Network 50: TRANSFER START_MFG TO STORAGE-2 WITH INLINE HOMO
   RUNG wire#powerrail
      { S7_Templates := "SrcType := Int" } EQ_Contact(in1 := "MODE SELECTION DB"."MODE BUFF", in2 := 1)
      { S7_Templates := "SrcType := Int" } EQ_Contact(in1 := "MFG TRANSFER CYCLE DB".TRANSFER."TRANSFER BUFF"."MFG TO STORAGE-2 WITH INLINE HOMO", in2 := 5)
      Coil( "AUTO ALARM DB"."MFG TRANSFER START"."MFG TO STORAGE-2 WITH INLINE HOMO" )
   END_RUNG
   // the same network as SCL:
   "AUTO ALARM DB"."MFG TRANSFER START"."MFG TO STORAGE-2 WITH INLINE HOMO" := ("MODE SELECTION DB"."MODE BUFF" = 1) AND ("MFG TRANSFER CYCLE DB".TRANSFER."TRANSFER BUFF"."MFG TO STORAGE-2 WITH INLINE HOMO" = 5);
END_REGION

REGION Network 51: TRANSFER OVER_MFG TO STORAGE-2 WITH INLINE HOMO
   RUNG wire#powerrail
      { S7_Templates := "SrcType := Int" } EQ_Contact(in1 := "MODE SELECTION DB"."MODE BUFF", in2 := 1)
      { S7_Templates := "SrcType := Int" } EQ_Contact(in1 := "MFG TRANSFER CYCLE DB".TRANSFER."TRANSFER BUFF"."MFG TO STORAGE-2 WITH INLINE HOMO", in2 := 15)
      Coil( "AUTO ALARM DB"."MFG TRANSFER OVER"."MFG TO STORAGE-2 WITH INLINE HOMO" )
   END_RUNG
   // the same network as SCL:
   "AUTO ALARM DB"."MFG TRANSFER OVER"."MFG TO STORAGE-2 WITH INLINE HOMO" := ("MODE SELECTION DB"."MODE BUFF" = 1) AND ("MFG TRANSFER CYCLE DB".TRANSFER."TRANSFER BUFF"."MFG TO STORAGE-2 WITH INLINE HOMO" = 15);
END_REGION

REGION Network 52: TRANSFER START_MFG TO STORAGE-2 WITH INLINE FILTER PRES
   RUNG wire#powerrail
      { S7_Templates := "SrcType := Int" } EQ_Contact(in1 := "MODE SELECTION DB"."MODE BUFF", in2 := 1)
      { S7_Templates := "SrcType := Int" } EQ_Contact(in1 := "MFG TRANSFER CYCLE DB".TRANSFER."TRANSFER BUFF"."MFG TO STORAGE-2 WITH INLINE FILTER PRES", in2 := 5)
      Coil( "AUTO ALARM DB"."MFG TRANSFER START"."MFG TO STORAGE-2 WITH INLINE FILTER PRES" )
   END_RUNG
   // the same network as SCL:
   "AUTO ALARM DB"."MFG TRANSFER START"."MFG TO STORAGE-2 WITH INLINE FILTER PRES" := ("MODE SELECTION DB"."MODE BUFF" = 1) AND ("MFG TRANSFER CYCLE DB".TRANSFER."TRANSFER BUFF"."MFG TO STORAGE-2 WITH INLINE FILTER PRES" = 5);
END_REGION

REGION Network 53: TRANSFER OVER_MFG TO STORAGE-2 WITH INLINE FILTER PRES
   RUNG wire#powerrail
      { S7_Templates := "SrcType := Int" } EQ_Contact(in1 := "MODE SELECTION DB"."MODE BUFF", in2 := 1)
      { S7_Templates := "SrcType := Int" } EQ_Contact(in1 := "MFG TRANSFER CYCLE DB".TRANSFER."TRANSFER BUFF"."MFG TO STORAGE-2 WITH INLINE FILTER PRES", in2 := 15)
      Coil( "AUTO ALARM DB"."MFG TRANSFER OVER"."MFG TO STORAGE-2 WITH INLINE FILTER PRES" )
   END_RUNG
   // the same network as SCL:
   "AUTO ALARM DB"."MFG TRANSFER OVER"."MFG TO STORAGE-2 WITH INLINE FILTER PRES" := ("MODE SELECTION DB"."MODE BUFF" = 1) AND ("MFG TRANSFER CYCLE DB".TRANSFER."TRANSFER BUFF"."MFG TO STORAGE-2 WITH INLINE FILTER PRES" = 15);
END_REGION

REGION Network 54: TRANSFER START_MFG TO STORAGE-3 WITH INLINE HOMO
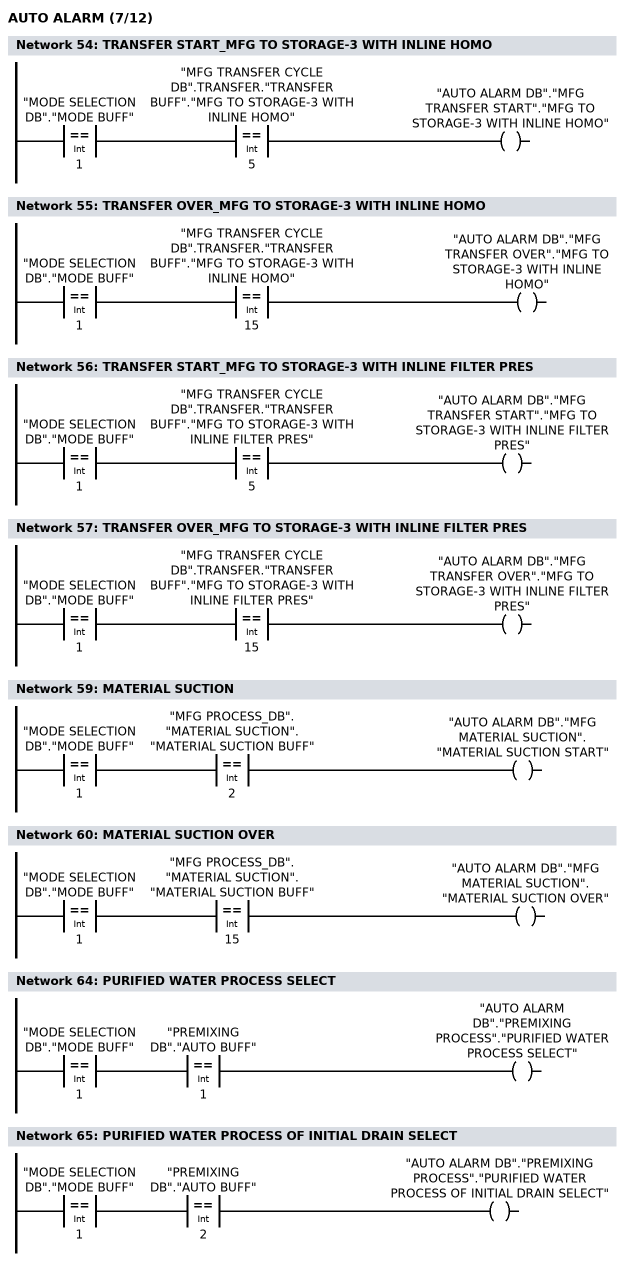
   RUNG wire#powerrail
      { S7_Templates := "SrcType := Int" } EQ_Contact(in1 := "MODE SELECTION DB"."MODE BUFF", in2 := 1)
      { S7_Templates := "SrcType := Int" } EQ_Contact(in1 := "MFG TRANSFER CYCLE DB".TRANSFER."TRANSFER BUFF"."MFG TO STORAGE-3 WITH INLINE HOMO", in2 := 5)
      Coil( "AUTO ALARM DB"."MFG TRANSFER START"."MFG TO STORAGE-3 WITH INLINE HOMO" )
   END_RUNG
   // the same network as SCL:
   "AUTO ALARM DB"."MFG TRANSFER START"."MFG TO STORAGE-3 WITH INLINE HOMO" := ("MODE SELECTION DB"."MODE BUFF" = 1) AND ("MFG TRANSFER CYCLE DB".TRANSFER."TRANSFER BUFF"."MFG TO STORAGE-3 WITH INLINE HOMO" = 5);
END_REGION

REGION Network 55: TRANSFER OVER_MFG TO STORAGE-3 WITH INLINE HOMO
   RUNG wire#powerrail
      { S7_Templates := "SrcType := Int" } EQ_Contact(in1 := "MODE SELECTION DB"."MODE BUFF", in2 := 1)
      { S7_Templates := "SrcType := Int" } EQ_Contact(in1 := "MFG TRANSFER CYCLE DB".TRANSFER."TRANSFER BUFF"."MFG TO STORAGE-3 WITH INLINE HOMO", in2 := 15)
      Coil( "AUTO ALARM DB"."MFG TRANSFER OVER"."MFG TO STORAGE-3 WITH INLINE HOMO" )
   END_RUNG
   // the same network as SCL:
   "AUTO ALARM DB"."MFG TRANSFER OVER"."MFG TO STORAGE-3 WITH INLINE HOMO" := ("MODE SELECTION DB"."MODE BUFF" = 1) AND ("MFG TRANSFER CYCLE DB".TRANSFER."TRANSFER BUFF"."MFG TO STORAGE-3 WITH INLINE HOMO" = 15);
END_REGION

REGION Network 56: TRANSFER START_MFG TO STORAGE-3 WITH INLINE FILTER PRES
   RUNG wire#powerrail
      { S7_Templates := "SrcType := Int" } EQ_Contact(in1 := "MODE SELECTION DB"."MODE BUFF", in2 := 1)
      { S7_Templates := "SrcType := Int" } EQ_Contact(in1 := "MFG TRANSFER CYCLE DB".TRANSFER."TRANSFER BUFF"."MFG TO STORAGE-3 WITH INLINE FILTER PRES", in2 := 5)
      Coil( "AUTO ALARM DB"."MFG TRANSFER START"."MFG TO STORAGE-3 WITH INLINE FILTER PRES" )
   END_RUNG
   // the same network as SCL:
   "AUTO ALARM DB"."MFG TRANSFER START"."MFG TO STORAGE-3 WITH INLINE FILTER PRES" := ("MODE SELECTION DB"."MODE BUFF" = 1) AND ("MFG TRANSFER CYCLE DB".TRANSFER."TRANSFER BUFF"."MFG TO STORAGE-3 WITH INLINE FILTER PRES" = 5);
END_REGION

REGION Network 57: TRANSFER OVER_MFG TO STORAGE-3 WITH INLINE FILTER PRES
   RUNG wire#powerrail
      { S7_Templates := "SrcType := Int" } EQ_Contact(in1 := "MODE SELECTION DB"."MODE BUFF", in2 := 1)
      { S7_Templates := "SrcType := Int" } EQ_Contact(in1 := "MFG TRANSFER CYCLE DB".TRANSFER."TRANSFER BUFF"."MFG TO STORAGE-3 WITH INLINE FILTER PRES", in2 := 15)
      Coil( "AUTO ALARM DB"."MFG TRANSFER OVER"."MFG TO STORAGE-3 WITH INLINE FILTER PRES" )
   END_RUNG
   // the same network as SCL:
   "AUTO ALARM DB"."MFG TRANSFER OVER"."MFG TO STORAGE-3 WITH INLINE FILTER PRES" := ("MODE SELECTION DB"."MODE BUFF" = 1) AND ("MFG TRANSFER CYCLE DB".TRANSFER."TRANSFER BUFF"."MFG TO STORAGE-3 WITH INLINE FILTER PRES" = 15);
END_REGION

REGION Network 59: MATERIAL SUCTION
   RUNG wire#powerrail
      { S7_Templates := "SrcType := Int" } EQ_Contact(in1 := "MODE SELECTION DB"."MODE BUFF", in2 := 1)
      { S7_Templates := "SrcType := Int" } EQ_Contact(in1 := "MFG PROCESS_DB"."MATERIAL SUCTION"."MATERIAL SUCTION BUFF", in2 := 2)
      Coil( "AUTO ALARM DB"."MFG MATERIAL SUCTION"."MATERIAL SUCTION START" )
   END_RUNG
   // the same network as SCL:
   "AUTO ALARM DB"."MFG MATERIAL SUCTION"."MATERIAL SUCTION START" := ("MODE SELECTION DB"."MODE BUFF" = 1) AND ("MFG PROCESS_DB"."MATERIAL SUCTION"."MATERIAL SUCTION BUFF" = 2);
END_REGION

REGION Network 60: MATERIAL SUCTION OVER
   RUNG wire#powerrail
      { S7_Templates := "SrcType := Int" } EQ_Contact(in1 := "MODE SELECTION DB"."MODE BUFF", in2 := 1)
      { S7_Templates := "SrcType := Int" } EQ_Contact(in1 := "MFG PROCESS_DB"."MATERIAL SUCTION"."MATERIAL SUCTION BUFF", in2 := 15)
      Coil( "AUTO ALARM DB"."MFG MATERIAL SUCTION"."MATERIAL SUCTION OVER" )
   END_RUNG
   // the same network as SCL:
   "AUTO ALARM DB"."MFG MATERIAL SUCTION"."MATERIAL SUCTION OVER" := ("MODE SELECTION DB"."MODE BUFF" = 1) AND ("MFG PROCESS_DB"."MATERIAL SUCTION"."MATERIAL SUCTION BUFF" = 15);
END_REGION

REGION Network 63: /////////////////////////////// PREMIXING PUPUP /////////////////////////////////////
END_REGION

REGION Network 64: PURIFIED WATER PROCESS SELECT
   RUNG wire#powerrail
      { S7_Templates := "SrcType := Int" } EQ_Contact(in1 := "MODE SELECTION DB"."MODE BUFF", in2 := 1)
      { S7_Templates := "SrcType := Int" } EQ_Contact(in1 := "PREMIXING DB"."AUTO BUFF", in2 := 1)
      Coil( "AUTO ALARM DB"."PREMIXING PROCESS"."PURIFIED WATER PROCESS SELECT" )
   END_RUNG
   // the same network as SCL:
   "AUTO ALARM DB"."PREMIXING PROCESS"."PURIFIED WATER PROCESS SELECT" := ("MODE SELECTION DB"."MODE BUFF" = 1) AND ("PREMIXING DB"."AUTO BUFF" = 1);
END_REGION

REGION Network 65: PURIFIED WATER PROCESS OF INITIAL DRAIN SELECT
   RUNG wire#powerrail
      { S7_Templates := "SrcType := Int" } EQ_Contact(in1 := "MODE SELECTION DB"."MODE BUFF", in2 := 1)
      { S7_Templates := "SrcType := Int" } EQ_Contact(in1 := "PREMIXING DB"."AUTO BUFF", in2 := 2)
      Coil( "AUTO ALARM DB"."PREMIXING PROCESS"."PURIFIED WATER PROCESS OF INITIAL DRAIN SELECT" )
   END_RUNG
   // the same network as SCL:
   "AUTO ALARM DB"."PREMIXING PROCESS"."PURIFIED WATER PROCESS OF INITIAL DRAIN SELECT" := ("MODE SELECTION DB"."MODE BUFF" = 1) AND ("PREMIXING DB"."AUTO BUFF" = 2);
END_REGION

REGION Network 66: PURIFIED WATER PROCESS OF LOAD CELL
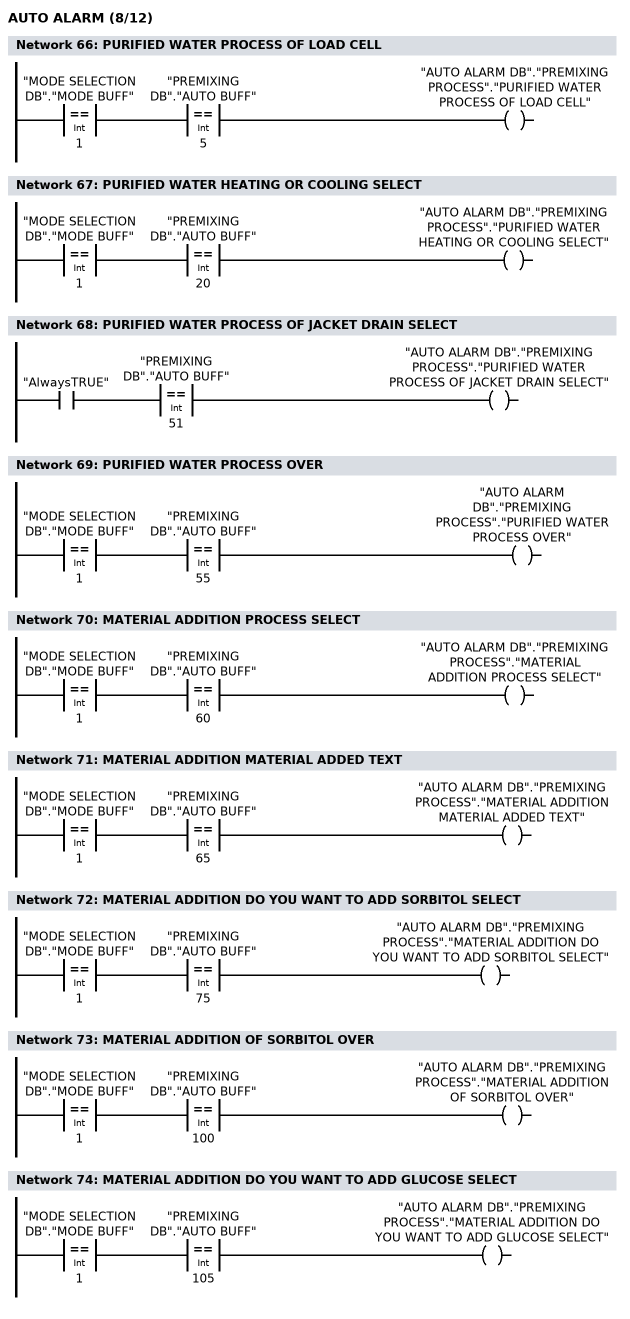
   RUNG wire#powerrail
      { S7_Templates := "SrcType := Int" } EQ_Contact(in1 := "MODE SELECTION DB"."MODE BUFF", in2 := 1)
      { S7_Templates := "SrcType := Int" } EQ_Contact(in1 := "PREMIXING DB"."AUTO BUFF", in2 := 5)
      Coil( "AUTO ALARM DB"."PREMIXING PROCESS"."PURIFIED WATER PROCESS OF LOAD CELL" )
   END_RUNG
   // the same network as SCL:
   "AUTO ALARM DB"."PREMIXING PROCESS"."PURIFIED WATER PROCESS OF LOAD CELL" := ("MODE SELECTION DB"."MODE BUFF" = 1) AND ("PREMIXING DB"."AUTO BUFF" = 5);
END_REGION

REGION Network 67: PURIFIED WATER HEATING OR COOLING SELECT
   RUNG wire#powerrail
      { S7_Templates := "SrcType := Int" } EQ_Contact(in1 := "MODE SELECTION DB"."MODE BUFF", in2 := 1)
      { S7_Templates := "SrcType := Int" } EQ_Contact(in1 := "PREMIXING DB"."AUTO BUFF", in2 := 20)
      Coil( "AUTO ALARM DB"."PREMIXING PROCESS"."PURIFIED WATER HEATING OR COOLING SELECT" )
   END_RUNG
   // the same network as SCL:
   "AUTO ALARM DB"."PREMIXING PROCESS"."PURIFIED WATER HEATING OR COOLING SELECT" := ("MODE SELECTION DB"."MODE BUFF" = 1) AND ("PREMIXING DB"."AUTO BUFF" = 20);
END_REGION

REGION Network 68: PURIFIED WATER PROCESS OF JACKET DRAIN SELECT
   RUNG wire#powerrail
      Contact( "AlwaysTRUE" )
      { S7_Templates := "SrcType := Int" } EQ_Contact(in1 := "PREMIXING DB"."AUTO BUFF", in2 := 51)
      Coil( "AUTO ALARM DB"."PREMIXING PROCESS"."PURIFIED WATER PROCESS OF JACKET DRAIN SELECT" )
   END_RUNG
   // the same network as SCL:
   "AUTO ALARM DB"."PREMIXING PROCESS"."PURIFIED WATER PROCESS OF JACKET DRAIN SELECT" := "AlwaysTRUE" AND ("PREMIXING DB"."AUTO BUFF" = 51);
END_REGION

REGION Network 69: PURIFIED WATER PROCESS OVER
   RUNG wire#powerrail
      { S7_Templates := "SrcType := Int" } EQ_Contact(in1 := "MODE SELECTION DB"."MODE BUFF", in2 := 1)
      { S7_Templates := "SrcType := Int" } EQ_Contact(in1 := "PREMIXING DB"."AUTO BUFF", in2 := 55)
      Coil( "AUTO ALARM DB"."PREMIXING PROCESS"."PURIFIED WATER PROCESS OVER" )
   END_RUNG
   // the same network as SCL:
   "AUTO ALARM DB"."PREMIXING PROCESS"."PURIFIED WATER PROCESS OVER" := ("MODE SELECTION DB"."MODE BUFF" = 1) AND ("PREMIXING DB"."AUTO BUFF" = 55);
END_REGION

REGION Network 70: MATERIAL ADDITION PROCESS SELECT
   RUNG wire#powerrail
      { S7_Templates := "SrcType := Int" } EQ_Contact(in1 := "MODE SELECTION DB"."MODE BUFF", in2 := 1)
      { S7_Templates := "SrcType := Int" } EQ_Contact(in1 := "PREMIXING DB"."AUTO BUFF", in2 := 60)
      Coil( "AUTO ALARM DB"."PREMIXING PROCESS"."MATERIAL ADDITION PROCESS SELECT" )
   END_RUNG
   // the same network as SCL:
   "AUTO ALARM DB"."PREMIXING PROCESS"."MATERIAL ADDITION PROCESS SELECT" := ("MODE SELECTION DB"."MODE BUFF" = 1) AND ("PREMIXING DB"."AUTO BUFF" = 60);
END_REGION

REGION Network 71: MATERIAL ADDITION MATERIAL ADDED TEXT
   RUNG wire#powerrail
      { S7_Templates := "SrcType := Int" } EQ_Contact(in1 := "MODE SELECTION DB"."MODE BUFF", in2 := 1)
      { S7_Templates := "SrcType := Int" } EQ_Contact(in1 := "PREMIXING DB"."AUTO BUFF", in2 := 65)
      Coil( "AUTO ALARM DB"."PREMIXING PROCESS"."MATERIAL ADDITION MATERIAL ADDED TEXT" )
   END_RUNG
   // the same network as SCL:
   "AUTO ALARM DB"."PREMIXING PROCESS"."MATERIAL ADDITION MATERIAL ADDED TEXT" := ("MODE SELECTION DB"."MODE BUFF" = 1) AND ("PREMIXING DB"."AUTO BUFF" = 65);
END_REGION

REGION Network 72: MATERIAL ADDITION DO YOU WANT TO ADD SORBITOL SELECT
   RUNG wire#powerrail
      { S7_Templates := "SrcType := Int" } EQ_Contact(in1 := "MODE SELECTION DB"."MODE BUFF", in2 := 1)
      { S7_Templates := "SrcType := Int" } EQ_Contact(in1 := "PREMIXING DB"."AUTO BUFF", in2 := 75)
      Coil( "AUTO ALARM DB"."PREMIXING PROCESS"."MATERIAL ADDITION DO YOU WANT TO ADD SORBITOL SELECT" )
   END_RUNG
   // the same network as SCL:
   "AUTO ALARM DB"."PREMIXING PROCESS"."MATERIAL ADDITION DO YOU WANT TO ADD SORBITOL SELECT" := ("MODE SELECTION DB"."MODE BUFF" = 1) AND ("PREMIXING DB"."AUTO BUFF" = 75);
END_REGION

REGION Network 73: MATERIAL ADDITION OF SORBITOL OVER
   RUNG wire#powerrail
      { S7_Templates := "SrcType := Int" } EQ_Contact(in1 := "MODE SELECTION DB"."MODE BUFF", in2 := 1)
      { S7_Templates := "SrcType := Int" } EQ_Contact(in1 := "PREMIXING DB"."AUTO BUFF", in2 := 100)
      Coil( "AUTO ALARM DB"."PREMIXING PROCESS"."MATERIAL ADDITION OF SORBITOL OVER" )
   END_RUNG
   // the same network as SCL:
   "AUTO ALARM DB"."PREMIXING PROCESS"."MATERIAL ADDITION OF SORBITOL OVER" := ("MODE SELECTION DB"."MODE BUFF" = 1) AND ("PREMIXING DB"."AUTO BUFF" = 100);
END_REGION

REGION Network 74: MATERIAL ADDITION DO YOU WANT TO ADD GLUCOSE SELECT
   RUNG wire#powerrail
      { S7_Templates := "SrcType := Int" } EQ_Contact(in1 := "MODE SELECTION DB"."MODE BUFF", in2 := 1)
      { S7_Templates := "SrcType := Int" } EQ_Contact(in1 := "PREMIXING DB"."AUTO BUFF", in2 := 105)
      Coil( "AUTO ALARM DB"."PREMIXING PROCESS"."MATERIAL ADDITION DO YOU WANT TO ADD GLUCOSE SELECT" )
   END_RUNG
   // the same network as SCL:
   "AUTO ALARM DB"."PREMIXING PROCESS"."MATERIAL ADDITION DO YOU WANT TO ADD GLUCOSE SELECT" := ("MODE SELECTION DB"."MODE BUFF" = 1) AND ("PREMIXING DB"."AUTO BUFF" = 105);
END_REGION

REGION Network 75: MATERIAL ADDITION OF GLUCOSE OVER
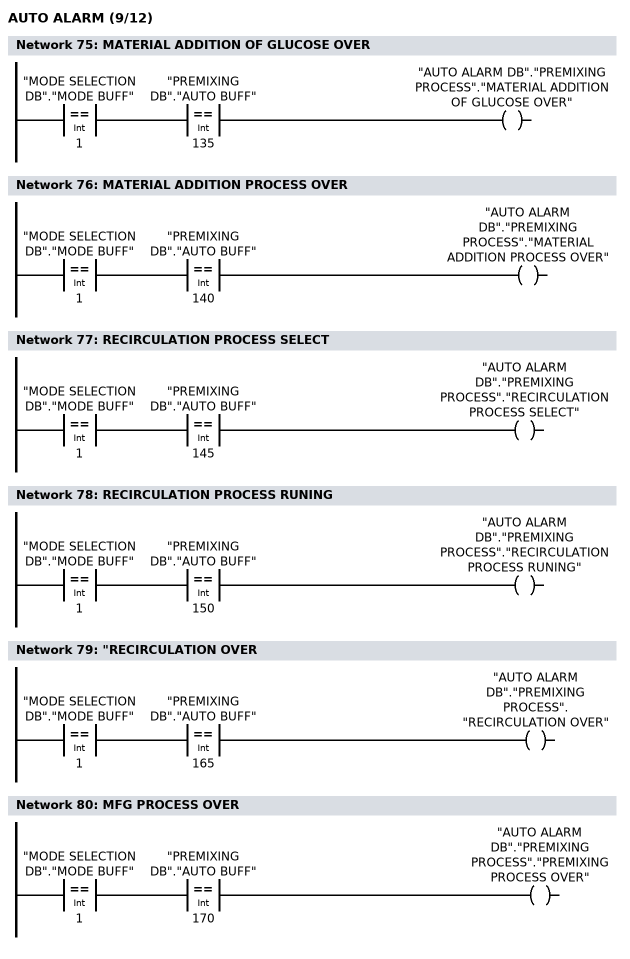
   RUNG wire#powerrail
      { S7_Templates := "SrcType := Int" } EQ_Contact(in1 := "MODE SELECTION DB"."MODE BUFF", in2 := 1)
      { S7_Templates := "SrcType := Int" } EQ_Contact(in1 := "PREMIXING DB"."AUTO BUFF", in2 := 135)
      Coil( "AUTO ALARM DB"."PREMIXING PROCESS"."MATERIAL ADDITION OF GLUCOSE OVER" )
   END_RUNG
   // the same network as SCL:
   "AUTO ALARM DB"."PREMIXING PROCESS"."MATERIAL ADDITION OF GLUCOSE OVER" := ("MODE SELECTION DB"."MODE BUFF" = 1) AND ("PREMIXING DB"."AUTO BUFF" = 135);
END_REGION

REGION Network 76: MATERIAL ADDITION PROCESS OVER
   RUNG wire#powerrail
      { S7_Templates := "SrcType := Int" } EQ_Contact(in1 := "MODE SELECTION DB"."MODE BUFF", in2 := 1)
      { S7_Templates := "SrcType := Int" } EQ_Contact(in1 := "PREMIXING DB"."AUTO BUFF", in2 := 140)
      Coil( "AUTO ALARM DB"."PREMIXING PROCESS"."MATERIAL ADDITION PROCESS OVER" )
   END_RUNG
   // the same network as SCL:
   "AUTO ALARM DB"."PREMIXING PROCESS"."MATERIAL ADDITION PROCESS OVER" := ("MODE SELECTION DB"."MODE BUFF" = 1) AND ("PREMIXING DB"."AUTO BUFF" = 140);
END_REGION

REGION Network 77: RECIRCULATION PROCESS SELECT
   RUNG wire#powerrail
      { S7_Templates := "SrcType := Int" } EQ_Contact(in1 := "MODE SELECTION DB"."MODE BUFF", in2 := 1)
      { S7_Templates := "SrcType := Int" } EQ_Contact(in1 := "PREMIXING DB"."AUTO BUFF", in2 := 145)
      Coil( "AUTO ALARM DB"."PREMIXING PROCESS"."RECIRCULATION PROCESS SELECT" )
   END_RUNG
   // the same network as SCL:
   "AUTO ALARM DB"."PREMIXING PROCESS"."RECIRCULATION PROCESS SELECT" := ("MODE SELECTION DB"."MODE BUFF" = 1) AND ("PREMIXING DB"."AUTO BUFF" = 145);
END_REGION

REGION Network 78: RECIRCULATION PROCESS RUNING
   RUNG wire#powerrail
      { S7_Templates := "SrcType := Int" } EQ_Contact(in1 := "MODE SELECTION DB"."MODE BUFF", in2 := 1)
      { S7_Templates := "SrcType := Int" } EQ_Contact(in1 := "PREMIXING DB"."AUTO BUFF", in2 := 150)
      Coil( "AUTO ALARM DB"."PREMIXING PROCESS"."RECIRCULATION PROCESS RUNING" )
   END_RUNG
   // the same network as SCL:
   "AUTO ALARM DB"."PREMIXING PROCESS"."RECIRCULATION PROCESS RUNING" := ("MODE SELECTION DB"."MODE BUFF" = 1) AND ("PREMIXING DB"."AUTO BUFF" = 150);
END_REGION

REGION Network 79: "RECIRCULATION OVER
   RUNG wire#powerrail
      { S7_Templates := "SrcType := Int" } EQ_Contact(in1 := "MODE SELECTION DB"."MODE BUFF", in2 := 1)
      { S7_Templates := "SrcType := Int" } EQ_Contact(in1 := "PREMIXING DB"."AUTO BUFF", in2 := 165)
      Coil( "AUTO ALARM DB"."PREMIXING PROCESS"."RECIRCULATION OVER" )
   END_RUNG
   // the same network as SCL:
   "AUTO ALARM DB"."PREMIXING PROCESS"."RECIRCULATION OVER" := ("MODE SELECTION DB"."MODE BUFF" = 1) AND ("PREMIXING DB"."AUTO BUFF" = 165);
END_REGION

REGION Network 80: MFG PROCESS OVER
   RUNG wire#powerrail
      { S7_Templates := "SrcType := Int" } EQ_Contact(in1 := "MODE SELECTION DB"."MODE BUFF", in2 := 1)
      { S7_Templates := "SrcType := Int" } EQ_Contact(in1 := "PREMIXING DB"."AUTO BUFF", in2 := 170)
      Coil( "AUTO ALARM DB"."PREMIXING PROCESS"."PREMIXING PROCESS OVER" )
   END_RUNG
   // the same network as SCL:
   "AUTO ALARM DB"."PREMIXING PROCESS"."PREMIXING PROCESS OVER" := ("MODE SELECTION DB"."MODE BUFF" = 1) AND ("PREMIXING DB"."AUTO BUFF" = 170);
END_REGION

REGION Network 82: PREMIXING TO MFG & STORAGE ALL IN ONE FOR OVER (POPUP)
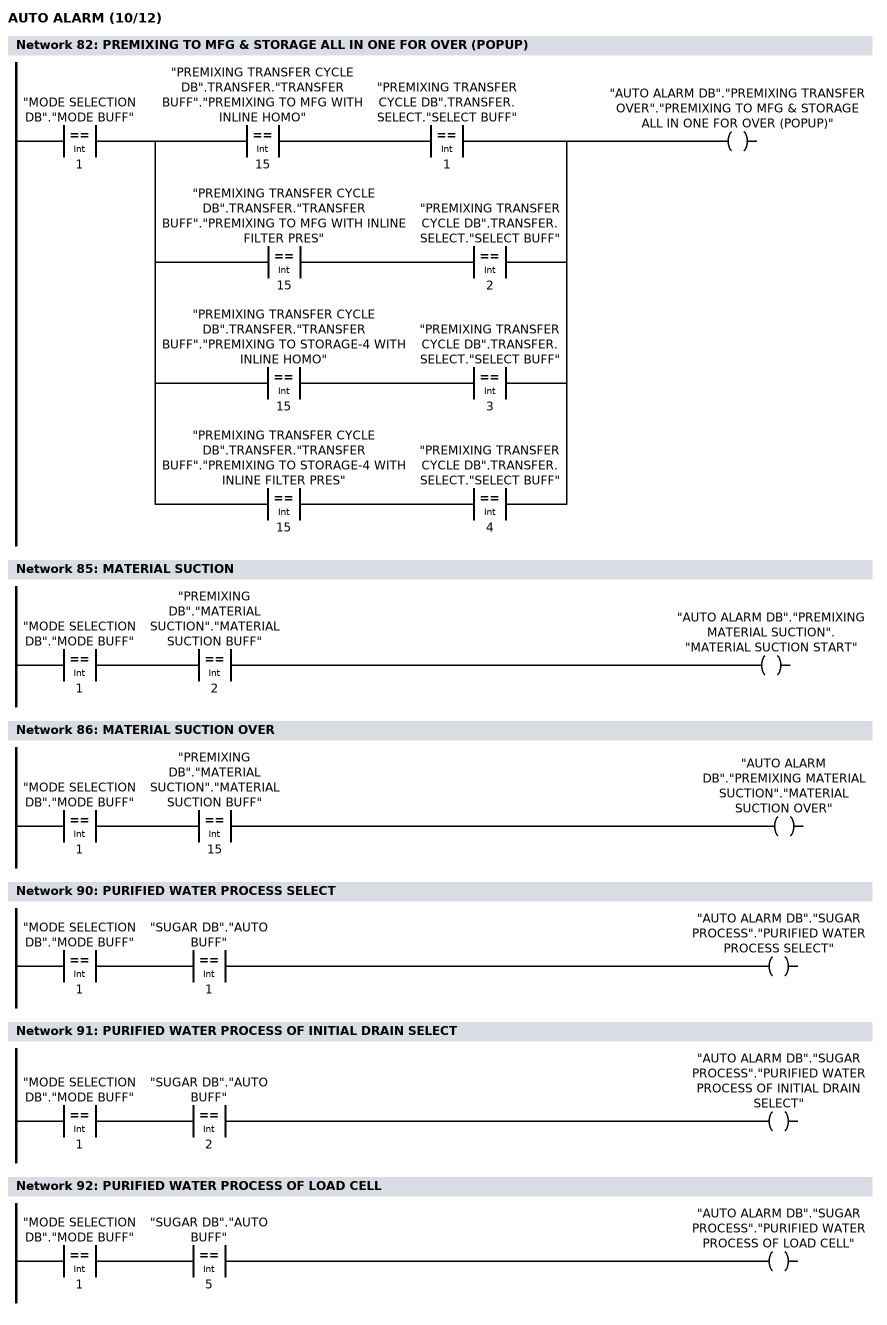
   RUNG wire#powerrail
      { S7_Templates := "SrcType := Int" } EQ_Contact(in1 := "MODE SELECTION DB"."MODE BUFF", in2 := 1)
      wire#w1
      { S7_Templates := "SrcType := Int" } EQ_Contact(in1 := "PREMIXING TRANSFER CYCLE DB".TRANSFER."TRANSFER BUFF"."PREMIXING TO MFG WITH INLINE HOMO", in2 := 15)
      { S7_Templates := "SrcType := Int" } EQ_Contact(in1 := "PREMIXING TRANSFER CYCLE DB".TRANSFER.SELECT."SELECT BUFF", in2 := 1)
      wire#w2
      Coil( "AUTO ALARM DB"."PREMIXING TRANSFER OVER"."PREMIXING TO MFG & STORAGE ALL IN ONE FOR OVER (POPUP)" )
   END_RUNG
   RUNG wire#w1
      { S7_Templates := "SrcType := Int" } EQ_Contact(in1 := "PREMIXING TRANSFER CYCLE DB".TRANSFER."TRANSFER BUFF"."PREMIXING TO MFG WITH INLINE FILTER PRES", in2 := 15)
      { S7_Templates := "SrcType := Int" } EQ_Contact(in1 := "PREMIXING TRANSFER CYCLE DB".TRANSFER.SELECT."SELECT BUFF", in2 := 2)
   END_RUNG wire#w2
   RUNG wire#w1
      { S7_Templates := "SrcType := Int" } EQ_Contact(in1 := "PREMIXING TRANSFER CYCLE DB".TRANSFER."TRANSFER BUFF"."PREMIXING TO STORAGE-4 WITH INLINE HOMO", in2 := 15)
      { S7_Templates := "SrcType := Int" } EQ_Contact(in1 := "PREMIXING TRANSFER CYCLE DB".TRANSFER.SELECT."SELECT BUFF", in2 := 3)
   END_RUNG wire#w2
   RUNG wire#w1
      { S7_Templates := "SrcType := Int" } EQ_Contact(in1 := "PREMIXING TRANSFER CYCLE DB".TRANSFER."TRANSFER BUFF"."PREMIXING TO STORAGE-4 WITH INLINE FILTER PRES", in2 := 15)
      { S7_Templates := "SrcType := Int" } EQ_Contact(in1 := "PREMIXING TRANSFER CYCLE DB".TRANSFER.SELECT."SELECT BUFF", in2 := 4)
   END_RUNG wire#w2
   // the same network as SCL:
   "AUTO ALARM DB"."PREMIXING TRANSFER OVER"."PREMIXING TO MFG & STORAGE ALL IN ONE FOR OVER (POPUP)" := ("MODE SELECTION DB"."MODE BUFF" = 1) AND ((("PREMIXING TRANSFER CYCLE DB".TRANSFER."TRANSFER BUFF"."PREMIXING TO MFG WITH INLINE HOMO" = 15) AND ("PREMIXING TRANSFER CYCLE DB".TRANSFER.SELECT."SELECT BUFF" = 1)) OR (("PREMIXING TRANSFER CYCLE DB".TRANSFER."TRANSFER BUFF"."PREMIXING TO MFG WITH INLINE FILTER PRES" = 15) AND ("PREMIXING TRANSFER CYCLE DB".TRANSFER.SELECT."SELECT BUFF" = 2)) OR (("PREMIXING TRANSFER CYCLE DB".TRANSFER."TRANSFER BUFF"."PREMIXING TO STORAGE-4 WITH INLINE HOMO" = 15) AND ("PREMIXING TRANSFER CYCLE DB".TRANSFER.SELECT."SELECT BUFF" = 3)) OR (("PREMIXING TRANSFER CYCLE DB".TRANSFER."TRANSFER BUFF"."PREMIXING TO STORAGE-4 WITH INLINE FILTER PRES" = 15) AND ("PREMIXING TRANSFER CYCLE DB".TRANSFER.SELECT."SELECT BUFF" = 4)));
END_REGION

REGION Network 85: MATERIAL SUCTION
   RUNG wire#powerrail
      { S7_Templates := "SrcType := Int" } EQ_Contact(in1 := "MODE SELECTION DB"."MODE BUFF", in2 := 1)
      { S7_Templates := "SrcType := Int" } EQ_Contact(in1 := "PREMIXING DB"."MATERIAL SUCTION"."MATERIAL SUCTION BUFF", in2 := 2)
      Coil( "AUTO ALARM DB"."PREMIXING MATERIAL SUCTION"."MATERIAL SUCTION START" )
   END_RUNG
   // the same network as SCL:
   "AUTO ALARM DB"."PREMIXING MATERIAL SUCTION"."MATERIAL SUCTION START" := ("MODE SELECTION DB"."MODE BUFF" = 1) AND ("PREMIXING DB"."MATERIAL SUCTION"."MATERIAL SUCTION BUFF" = 2);
END_REGION

REGION Network 86: MATERIAL SUCTION OVER
   RUNG wire#powerrail
      { S7_Templates := "SrcType := Int" } EQ_Contact(in1 := "MODE SELECTION DB"."MODE BUFF", in2 := 1)
      { S7_Templates := "SrcType := Int" } EQ_Contact(in1 := "PREMIXING DB"."MATERIAL SUCTION"."MATERIAL SUCTION BUFF", in2 := 15)
      Coil( "AUTO ALARM DB"."PREMIXING MATERIAL SUCTION"."MATERIAL SUCTION OVER" )
   END_RUNG
   // the same network as SCL:
   "AUTO ALARM DB"."PREMIXING MATERIAL SUCTION"."MATERIAL SUCTION OVER" := ("MODE SELECTION DB"."MODE BUFF" = 1) AND ("PREMIXING DB"."MATERIAL SUCTION"."MATERIAL SUCTION BUFF" = 15);
END_REGION

REGION Network 89: /////////////////////////////// SUGAR PUPUP /////////////////////////////////////
END_REGION

REGION Network 90: PURIFIED WATER PROCESS SELECT
   RUNG wire#powerrail
      { S7_Templates := "SrcType := Int" } EQ_Contact(in1 := "MODE SELECTION DB"."MODE BUFF", in2 := 1)
      { S7_Templates := "SrcType := Int" } EQ_Contact(in1 := "SUGAR DB"."AUTO BUFF", in2 := 1)
      Coil( "AUTO ALARM DB"."SUGAR PROCESS"."PURIFIED WATER PROCESS SELECT" )
   END_RUNG
   // the same network as SCL:
   "AUTO ALARM DB"."SUGAR PROCESS"."PURIFIED WATER PROCESS SELECT" := ("MODE SELECTION DB"."MODE BUFF" = 1) AND ("SUGAR DB"."AUTO BUFF" = 1);
END_REGION

REGION Network 91: PURIFIED WATER PROCESS OF INITIAL DRAIN SELECT
   RUNG wire#powerrail
      { S7_Templates := "SrcType := Int" } EQ_Contact(in1 := "MODE SELECTION DB"."MODE BUFF", in2 := 1)
      { S7_Templates := "SrcType := Int" } EQ_Contact(in1 := "SUGAR DB"."AUTO BUFF", in2 := 2)
      Coil( "AUTO ALARM DB"."SUGAR PROCESS"."PURIFIED WATER PROCESS OF INITIAL DRAIN SELECT" )
   END_RUNG
   // the same network as SCL:
   "AUTO ALARM DB"."SUGAR PROCESS"."PURIFIED WATER PROCESS OF INITIAL DRAIN SELECT" := ("MODE SELECTION DB"."MODE BUFF" = 1) AND ("SUGAR DB"."AUTO BUFF" = 2);
END_REGION

REGION Network 92: PURIFIED WATER PROCESS OF LOAD CELL
   RUNG wire#powerrail
      { S7_Templates := "SrcType := Int" } EQ_Contact(in1 := "MODE SELECTION DB"."MODE BUFF", in2 := 1)
      { S7_Templates := "SrcType := Int" } EQ_Contact(in1 := "SUGAR DB"."AUTO BUFF", in2 := 5)
      Coil( "AUTO ALARM DB"."SUGAR PROCESS"."PURIFIED WATER PROCESS OF LOAD CELL" )
   END_RUNG
   // the same network as SCL:
   "AUTO ALARM DB"."SUGAR PROCESS"."PURIFIED WATER PROCESS OF LOAD CELL" := ("MODE SELECTION DB"."MODE BUFF" = 1) AND ("SUGAR DB"."AUTO BUFF" = 5);
END_REGION

REGION Network 93: PURIFIED WATER HEATING OR COOLING SELECT
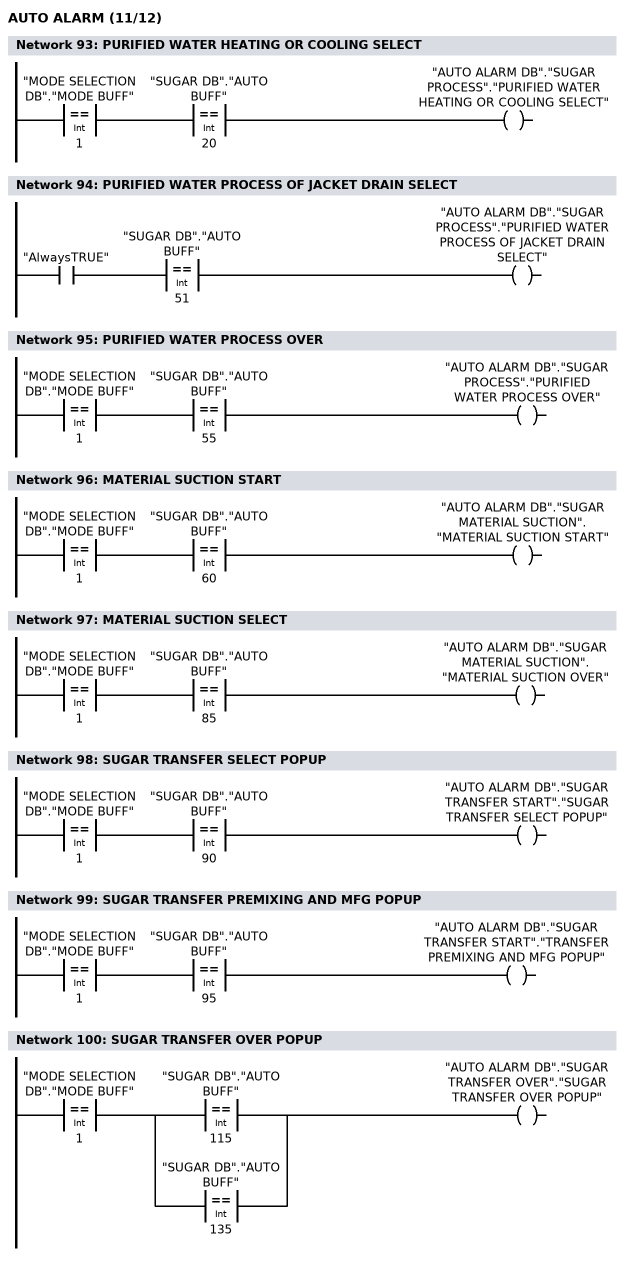
   RUNG wire#powerrail
      { S7_Templates := "SrcType := Int" } EQ_Contact(in1 := "MODE SELECTION DB"."MODE BUFF", in2 := 1)
      { S7_Templates := "SrcType := Int" } EQ_Contact(in1 := "SUGAR DB"."AUTO BUFF", in2 := 20)
      Coil( "AUTO ALARM DB"."SUGAR PROCESS"."PURIFIED WATER HEATING OR COOLING SELECT" )
   END_RUNG
   // the same network as SCL:
   "AUTO ALARM DB"."SUGAR PROCESS"."PURIFIED WATER HEATING OR COOLING SELECT" := ("MODE SELECTION DB"."MODE BUFF" = 1) AND ("SUGAR DB"."AUTO BUFF" = 20);
END_REGION

REGION Network 94: PURIFIED WATER PROCESS OF JACKET DRAIN SELECT
   RUNG wire#powerrail
      Contact( "AlwaysTRUE" )
      { S7_Templates := "SrcType := Int" } EQ_Contact(in1 := "SUGAR DB"."AUTO BUFF", in2 := 51)
      Coil( "AUTO ALARM DB"."SUGAR PROCESS"."PURIFIED WATER PROCESS OF JACKET DRAIN SELECT" )
   END_RUNG
   // the same network as SCL:
   "AUTO ALARM DB"."SUGAR PROCESS"."PURIFIED WATER PROCESS OF JACKET DRAIN SELECT" := "AlwaysTRUE" AND ("SUGAR DB"."AUTO BUFF" = 51);
END_REGION

REGION Network 95: PURIFIED WATER PROCESS OVER
   RUNG wire#powerrail
      { S7_Templates := "SrcType := Int" } EQ_Contact(in1 := "MODE SELECTION DB"."MODE BUFF", in2 := 1)
      { S7_Templates := "SrcType := Int" } EQ_Contact(in1 := "SUGAR DB"."AUTO BUFF", in2 := 55)
      Coil( "AUTO ALARM DB"."SUGAR PROCESS"."PURIFIED WATER PROCESS OVER" )
   END_RUNG
   // the same network as SCL:
   "AUTO ALARM DB"."SUGAR PROCESS"."PURIFIED WATER PROCESS OVER" := ("MODE SELECTION DB"."MODE BUFF" = 1) AND ("SUGAR DB"."AUTO BUFF" = 55);
END_REGION

REGION Network 96: MATERIAL SUCTION START
   RUNG wire#powerrail
      { S7_Templates := "SrcType := Int" } EQ_Contact(in1 := "MODE SELECTION DB"."MODE BUFF", in2 := 1)
      { S7_Templates := "SrcType := Int" } EQ_Contact(in1 := "SUGAR DB"."AUTO BUFF", in2 := 60)
      Coil( "AUTO ALARM DB"."SUGAR MATERIAL SUCTION"."MATERIAL SUCTION START" )
   END_RUNG
   // the same network as SCL:
   "AUTO ALARM DB"."SUGAR MATERIAL SUCTION"."MATERIAL SUCTION START" := ("MODE SELECTION DB"."MODE BUFF" = 1) AND ("SUGAR DB"."AUTO BUFF" = 60);
END_REGION

REGION Network 97: MATERIAL SUCTION SELECT
   RUNG wire#powerrail
      { S7_Templates := "SrcType := Int" } EQ_Contact(in1 := "MODE SELECTION DB"."MODE BUFF", in2 := 1)
      { S7_Templates := "SrcType := Int" } EQ_Contact(in1 := "SUGAR DB"."AUTO BUFF", in2 := 85)
      Coil( "AUTO ALARM DB"."SUGAR MATERIAL SUCTION"."MATERIAL SUCTION OVER" )
   END_RUNG
   // the same network as SCL:
   "AUTO ALARM DB"."SUGAR MATERIAL SUCTION"."MATERIAL SUCTION OVER" := ("MODE SELECTION DB"."MODE BUFF" = 1) AND ("SUGAR DB"."AUTO BUFF" = 85);
END_REGION

REGION Network 98: SUGAR TRANSFER SELECT POPUP
   RUNG wire#powerrail
      { S7_Templates := "SrcType := Int" } EQ_Contact(in1 := "MODE SELECTION DB"."MODE BUFF", in2 := 1)
      { S7_Templates := "SrcType := Int" } EQ_Contact(in1 := "SUGAR DB"."AUTO BUFF", in2 := 90)
      Coil( "AUTO ALARM DB"."SUGAR TRANSFER START"."SUGAR TRANSFER SELECT POPUP" )
   END_RUNG
   // the same network as SCL:
   "AUTO ALARM DB"."SUGAR TRANSFER START"."SUGAR TRANSFER SELECT POPUP" := ("MODE SELECTION DB"."MODE BUFF" = 1) AND ("SUGAR DB"."AUTO BUFF" = 90);
END_REGION

REGION Network 99: SUGAR TRANSFER PREMIXING AND MFG POPUP
   RUNG wire#powerrail
      { S7_Templates := "SrcType := Int" } EQ_Contact(in1 := "MODE SELECTION DB"."MODE BUFF", in2 := 1)
      { S7_Templates := "SrcType := Int" } EQ_Contact(in1 := "SUGAR DB"."AUTO BUFF", in2 := 95)
      Coil( "AUTO ALARM DB"."SUGAR TRANSFER START"."TRANSFER PREMIXING AND MFG POPUP" )
   END_RUNG
   // the same network as SCL:
   "AUTO ALARM DB"."SUGAR TRANSFER START"."TRANSFER PREMIXING AND MFG POPUP" := ("MODE SELECTION DB"."MODE BUFF" = 1) AND ("SUGAR DB"."AUTO BUFF" = 95);
END_REGION

REGION Network 100: SUGAR TRANSFER OVER POPUP
   RUNG wire#powerrail
      { S7_Templates := "SrcType := Int" } EQ_Contact(in1 := "MODE SELECTION DB"."MODE BUFF", in2 := 1)
      wire#w1
      { S7_Templates := "SrcType := Int" } EQ_Contact(in1 := "SUGAR DB"."AUTO BUFF", in2 := 115)
      wire#w2
      Coil( "AUTO ALARM DB"."SUGAR TRANSFER OVER"."SUGAR TRANSFER OVER POPUP" )
   END_RUNG
   RUNG wire#w1
      { S7_Templates := "SrcType := Int" } EQ_Contact(in1 := "SUGAR DB"."AUTO BUFF", in2 := 135)
   END_RUNG wire#w2
   // the same network as SCL:
   "AUTO ALARM DB"."SUGAR TRANSFER OVER"."SUGAR TRANSFER OVER POPUP" := ("MODE SELECTION DB"."MODE BUFF" = 1) AND (("SUGAR DB"."AUTO BUFF" = 115) OR ("SUGAR DB"."AUTO BUFF" = 135));
END_REGION

REGION Network 101: SUGAR PROCESS OVER
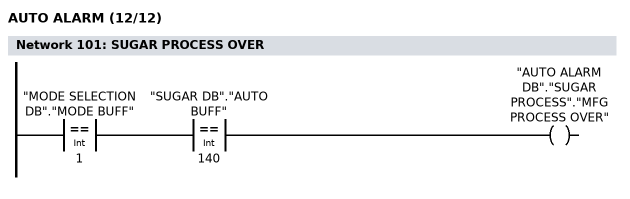
   RUNG wire#powerrail
      { S7_Templates := "SrcType := Int" } EQ_Contact(in1 := "MODE SELECTION DB"."MODE BUFF", in2 := 1)
      { S7_Templates := "SrcType := Int" } EQ_Contact(in1 := "SUGAR DB"."AUTO BUFF", in2 := 140)
      Coil( "AUTO ALARM DB"."SUGAR PROCESS"."MFG PROCESS OVER" )
   END_RUNG
   // the same network as SCL:
   "AUTO ALARM DB"."SUGAR PROCESS"."MFG PROCESS OVER" := ("MODE SELECTION DB"."MODE BUFF" = 1) AND ("SUGAR DB"."AUTO BUFF" = 140);
END_REGION
END_FUNCTION

FUNCTION "MANUAL INTERLOCK" : Void   // FC8, LAD
{ S7_Optimized_Access := 'TRUE' }
// stored: SetENOAutomatically false
BEGIN

REGION Network 1: ERROR BIT
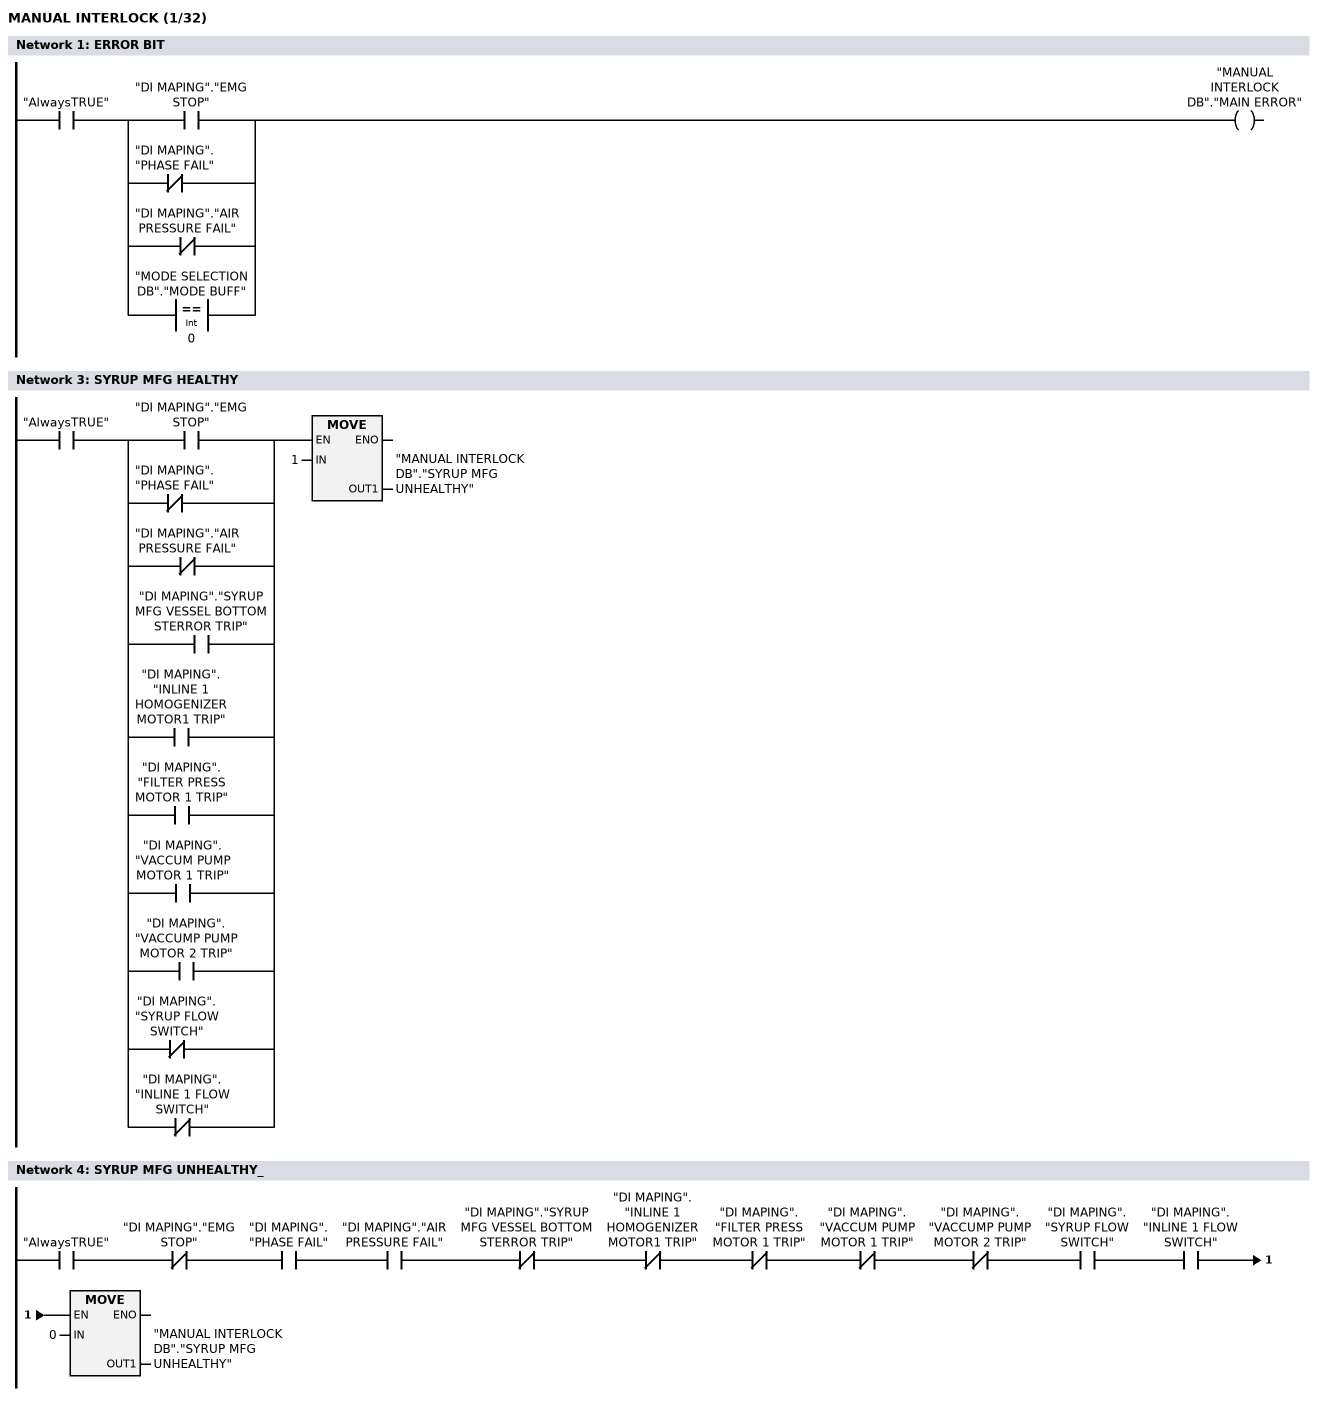
   RUNG wire#powerrail
      Contact( "AlwaysTRUE" )
      wire#w1
      Contact( "DI MAPING"."EMG STOP" )
      wire#w2
      Coil( "MANUAL INTERLOCK DB"."MAIN ERROR" )
   END_RUNG
   RUNG wire#w1
      I_Contact( "DI MAPING"."PHASE FAIL" )
   END_RUNG wire#w2
   RUNG wire#w1
      I_Contact( "DI MAPING"."AIR PRESSURE FAIL" )
   END_RUNG wire#w2
   RUNG wire#w1
      { S7_Templates := "SrcType := Int" } EQ_Contact(in1 := "MODE SELECTION DB"."MODE BUFF", in2 := 0)
   END_RUNG wire#w2
   // the same network as SCL:
   "MANUAL INTERLOCK DB"."MAIN ERROR" := "AlwaysTRUE" AND ("DI MAPING"."EMG STOP" OR NOT "DI MAPING"."PHASE FAIL" OR NOT "DI MAPING"."AIR PRESSURE FAIL" OR ("MODE SELECTION DB"."MODE BUFF" = 0));
END_REGION

REGION Network 3: SYRUP MFG HEALTHY
   RUNG wire#powerrail
      Contact( "AlwaysTRUE" )
      wire#w1
      Contact( "DI MAPING"."EMG STOP" )
      wire#w2
      Move(in := 1, out1 => "MANUAL INTERLOCK DB"."SYRUP MFG UNHEALTHY")
   END_RUNG
   RUNG wire#w1
      I_Contact( "DI MAPING"."PHASE FAIL" )
   END_RUNG wire#w2
   RUNG wire#w1
      I_Contact( "DI MAPING"."AIR PRESSURE FAIL" )
   END_RUNG wire#w2
   RUNG wire#w1
      Contact( "DI MAPING"."SYRUP MFG VESSEL BOTTOM STERROR TRIP" )
   END_RUNG wire#w2
   RUNG wire#w1
      Contact( "DI MAPING"."INLINE 1 HOMOGENIZER MOTOR1 TRIP" )
   END_RUNG wire#w2
   RUNG wire#w1
      Contact( "DI MAPING"."FILTER PRESS MOTOR 1 TRIP" )
   END_RUNG wire#w2
   RUNG wire#w1
      Contact( "DI MAPING"."VACCUM PUMP MOTOR 1 TRIP" )
   END_RUNG wire#w2
   RUNG wire#w1
      Contact( "DI MAPING"."VACCUMP PUMP MOTOR 2 TRIP" )
   END_RUNG wire#w2
   RUNG wire#w1
      I_Contact( "DI MAPING"."SYRUP FLOW SWITCH" )
   END_RUNG wire#w2
   RUNG wire#w1
      I_Contact( "DI MAPING"."INLINE 1 FLOW SWITCH" )
   END_RUNG wire#w2
   // the same network as SCL:
   IF "AlwaysTRUE" AND ("DI MAPING"."EMG STOP" OR NOT "DI MAPING"."PHASE FAIL" OR NOT "DI MAPING"."AIR PRESSURE FAIL" OR "DI MAPING"."SYRUP MFG VESSEL BOTTOM STERROR TRIP" OR "DI MAPING"."INLINE 1 HOMOGENIZER MOTOR1 TRIP" OR "DI MAPING"."FILTER PRESS MOTOR 1 TRIP" OR "DI MAPING"."VACCUM PUMP MOTOR 1 TRIP" OR "DI MAPING"."VACCUMP PUMP MOTOR 2 TRIP" OR NOT "DI MAPING"."SYRUP FLOW SWITCH" OR NOT "DI MAPING"."INLINE 1 FLOW SWITCH") THEN
       "MANUAL INTERLOCK DB"."SYRUP MFG UNHEALTHY" := 1;
   END_IF;
END_REGION

REGION Network 4: SYRUP MFG UNHEALTHY_
   RUNG wire#powerrail
      Contact( "AlwaysTRUE" )
      I_Contact( "DI MAPING"."EMG STOP" )
      Contact( "DI MAPING"."PHASE FAIL" )
      Contact( "DI MAPING"."AIR PRESSURE FAIL" )
      I_Contact( "DI MAPING"."SYRUP MFG VESSEL BOTTOM STERROR TRIP" )
      I_Contact( "DI MAPING"."INLINE 1 HOMOGENIZER MOTOR1 TRIP" )
      I_Contact( "DI MAPING"."FILTER PRESS MOTOR 1 TRIP" )
      I_Contact( "DI MAPING"."VACCUM PUMP MOTOR 1 TRIP" )
      I_Contact( "DI MAPING"."VACCUMP PUMP MOTOR 2 TRIP" )
      Contact( "DI MAPING"."SYRUP FLOW SWITCH" )
      Contact( "DI MAPING"."INLINE 1 FLOW SWITCH" )
      Move(in := 0, out1 => "MANUAL INTERLOCK DB"."SYRUP MFG UNHEALTHY")
   END_RUNG
   // the same network as SCL:
   IF "AlwaysTRUE" AND NOT "DI MAPING"."EMG STOP" AND "DI MAPING"."PHASE FAIL" AND "DI MAPING"."AIR PRESSURE FAIL" AND NOT "DI MAPING"."SYRUP MFG VESSEL BOTTOM STERROR TRIP" AND NOT "DI MAPING"."INLINE 1 HOMOGENIZER MOTOR1 TRIP" AND NOT "DI MAPING"."FILTER PRESS MOTOR 1 TRIP" AND NOT "DI MAPING"."VACCUM PUMP MOTOR 1 TRIP" AND NOT "DI MAPING"."VACCUMP PUMP MOTOR 2 TRIP" AND "DI MAPING"."SYRUP FLOW SWITCH" AND "DI MAPING"."INLINE 1 FLOW SWITCH" THEN
       "MANUAL INTERLOCK DB"."SYRUP MFG UNHEALTHY" := 0;
   END_IF;
END_REGION

REGION Network 5: PREMIXING HEALTHY
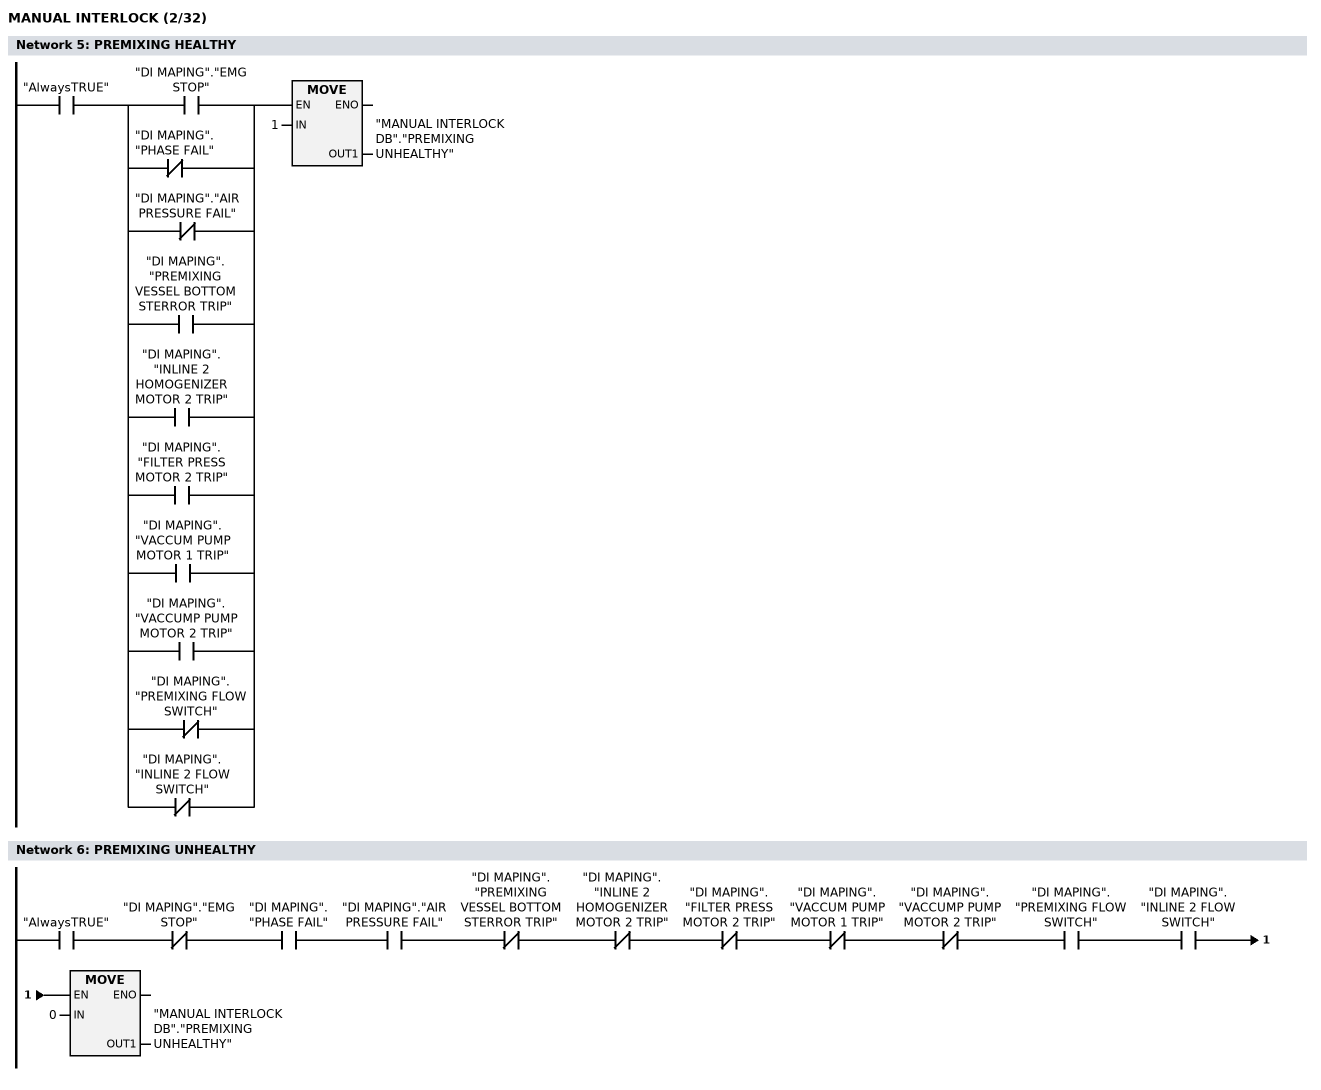
   RUNG wire#powerrail
      Contact( "AlwaysTRUE" )
      wire#w1
      Contact( "DI MAPING"."EMG STOP" )
      wire#w2
      Move(in := 1, out1 => "MANUAL INTERLOCK DB"."PREMIXING UNHEALTHY")
   END_RUNG
   RUNG wire#w1
      I_Contact( "DI MAPING"."PHASE FAIL" )
   END_RUNG wire#w2
   RUNG wire#w1
      I_Contact( "DI MAPING"."AIR PRESSURE FAIL" )
   END_RUNG wire#w2
   RUNG wire#w1
      Contact( "DI MAPING"."PREMIXING VESSEL BOTTOM STERROR TRIP" )
   END_RUNG wire#w2
   RUNG wire#w1
      Contact( "DI MAPING"."INLINE 2 HOMOGENIZER MOTOR 2 TRIP" )
   END_RUNG wire#w2
   RUNG wire#w1
      Contact( "DI MAPING"."FILTER PRESS MOTOR 2 TRIP" )
   END_RUNG wire#w2
   RUNG wire#w1
      Contact( "DI MAPING"."VACCUM PUMP MOTOR 1 TRIP" )
   END_RUNG wire#w2
   RUNG wire#w1
      Contact( "DI MAPING"."VACCUMP PUMP MOTOR 2 TRIP" )
   END_RUNG wire#w2
   RUNG wire#w1
      I_Contact( "DI MAPING"."PREMIXING FLOW SWITCH" )
   END_RUNG wire#w2
   RUNG wire#w1
      I_Contact( "DI MAPING"."INLINE 2 FLOW SWITCH" )
   END_RUNG wire#w2
   // the same network as SCL:
   IF "AlwaysTRUE" AND ("DI MAPING"."EMG STOP" OR NOT "DI MAPING"."PHASE FAIL" OR NOT "DI MAPING"."AIR PRESSURE FAIL" OR "DI MAPING"."PREMIXING VESSEL BOTTOM STERROR TRIP" OR "DI MAPING"."INLINE 2 HOMOGENIZER MOTOR 2 TRIP" OR "DI MAPING"."FILTER PRESS MOTOR 2 TRIP" OR "DI MAPING"."VACCUM PUMP MOTOR 1 TRIP" OR "DI MAPING"."VACCUMP PUMP MOTOR 2 TRIP" OR NOT "DI MAPING"."PREMIXING FLOW SWITCH" OR NOT "DI MAPING"."INLINE 2 FLOW SWITCH") THEN
       "MANUAL INTERLOCK DB"."PREMIXING UNHEALTHY" := 1;
   END_IF;
END_REGION

REGION Network 6: PREMIXING UNHEALTHY
   RUNG wire#powerrail
      Contact( "AlwaysTRUE" )
      I_Contact( "DI MAPING"."EMG STOP" )
      Contact( "DI MAPING"."PHASE FAIL" )
      Contact( "DI MAPING"."AIR PRESSURE FAIL" )
      I_Contact( "DI MAPING"."PREMIXING VESSEL BOTTOM STERROR TRIP" )
      I_Contact( "DI MAPING"."INLINE 2 HOMOGENIZER MOTOR 2 TRIP" )
      I_Contact( "DI MAPING"."FILTER PRESS MOTOR 2 TRIP" )
      I_Contact( "DI MAPING"."VACCUM PUMP MOTOR 1 TRIP" )
      I_Contact( "DI MAPING"."VACCUMP PUMP MOTOR 2 TRIP" )
      Contact( "DI MAPING"."PREMIXING FLOW SWITCH" )
      Contact( "DI MAPING"."INLINE 2 FLOW SWITCH" )
      Move(in := 0, out1 => "MANUAL INTERLOCK DB"."PREMIXING UNHEALTHY")
   END_RUNG
   // the same network as SCL:
   IF "AlwaysTRUE" AND NOT "DI MAPING"."EMG STOP" AND "DI MAPING"."PHASE FAIL" AND "DI MAPING"."AIR PRESSURE FAIL" AND NOT "DI MAPING"."PREMIXING VESSEL BOTTOM STERROR TRIP" AND NOT "DI MAPING"."INLINE 2 HOMOGENIZER MOTOR 2 TRIP" AND NOT "DI MAPING"."FILTER PRESS MOTOR 2 TRIP" AND NOT "DI MAPING"."VACCUM PUMP MOTOR 1 TRIP" AND NOT "DI MAPING"."VACCUMP PUMP MOTOR 2 TRIP" AND "DI MAPING"."PREMIXING FLOW SWITCH" AND "DI MAPING"."INLINE 2 FLOW SWITCH" THEN
       "MANUAL INTERLOCK DB"."PREMIXING UNHEALTHY" := 0;
   END_IF;
END_REGION

REGION Network 7: SUGAR HEALTHY
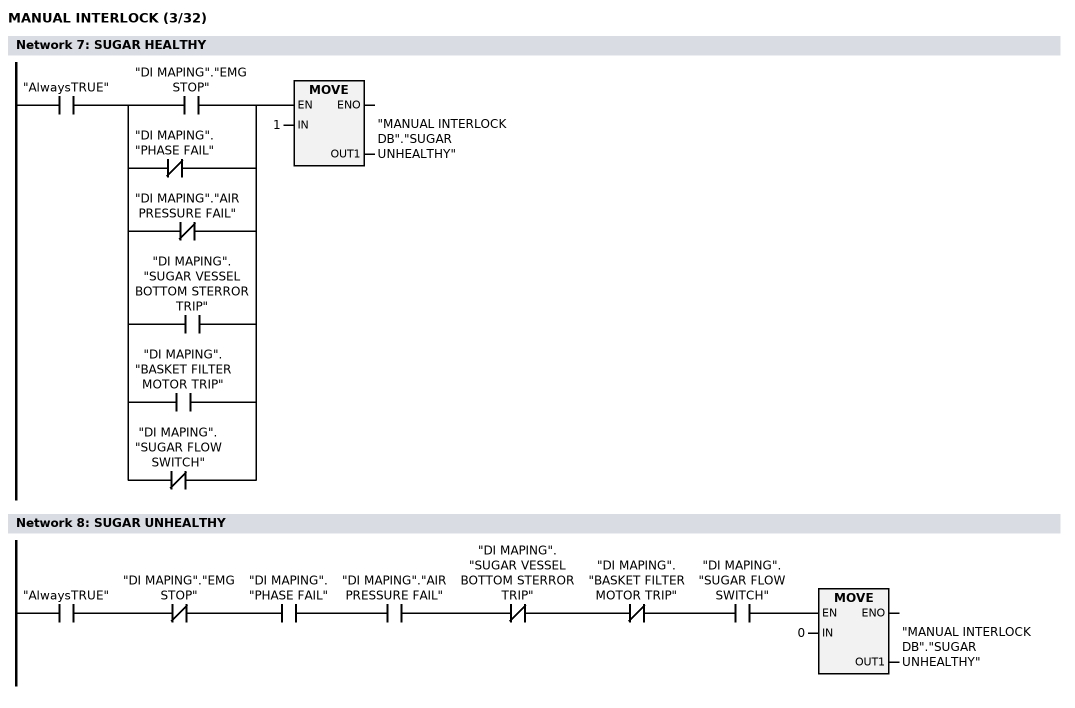
   RUNG wire#powerrail
      Contact( "AlwaysTRUE" )
      wire#w1
      Contact( "DI MAPING"."EMG STOP" )
      wire#w2
      Move(in := 1, out1 => "MANUAL INTERLOCK DB"."SUGAR UNHEALTHY")
   END_RUNG
   RUNG wire#w1
      I_Contact( "DI MAPING"."PHASE FAIL" )
   END_RUNG wire#w2
   RUNG wire#w1
      I_Contact( "DI MAPING"."AIR PRESSURE FAIL" )
   END_RUNG wire#w2
   RUNG wire#w1
      Contact( "DI MAPING"."SUGAR VESSEL BOTTOM STERROR TRIP" )
   END_RUNG wire#w2
   RUNG wire#w1
      Contact( "DI MAPING"."BASKET FILTER MOTOR TRIP" )
   END_RUNG wire#w2
   RUNG wire#w1
      I_Contact( "DI MAPING"."SUGAR FLOW SWITCH" )
   END_RUNG wire#w2
   // the same network as SCL:
   IF "AlwaysTRUE" AND ("DI MAPING"."EMG STOP" OR NOT "DI MAPING"."PHASE FAIL" OR NOT "DI MAPING"."AIR PRESSURE FAIL" OR "DI MAPING"."SUGAR VESSEL BOTTOM STERROR TRIP" OR "DI MAPING"."BASKET FILTER MOTOR TRIP" OR NOT "DI MAPING"."SUGAR FLOW SWITCH") THEN
       "MANUAL INTERLOCK DB"."SUGAR UNHEALTHY" := 1;
   END_IF;
END_REGION

REGION Network 8: SUGAR UNHEALTHY
   RUNG wire#powerrail
      Contact( "AlwaysTRUE" )
      I_Contact( "DI MAPING"."EMG STOP" )
      Contact( "DI MAPING"."PHASE FAIL" )
      Contact( "DI MAPING"."AIR PRESSURE FAIL" )
      I_Contact( "DI MAPING"."SUGAR VESSEL BOTTOM STERROR TRIP" )
      I_Contact( "DI MAPING"."BASKET FILTER MOTOR TRIP" )
      Contact( "DI MAPING"."SUGAR FLOW SWITCH" )
      Move(in := 0, out1 => "MANUAL INTERLOCK DB"."SUGAR UNHEALTHY")
   END_RUNG
   // the same network as SCL:
   IF "AlwaysTRUE" AND NOT "DI MAPING"."EMG STOP" AND "DI MAPING"."PHASE FAIL" AND "DI MAPING"."AIR PRESSURE FAIL" AND NOT "DI MAPING"."SUGAR VESSEL BOTTOM STERROR TRIP" AND NOT "DI MAPING"."BASKET FILTER MOTOR TRIP" AND "DI MAPING"."SUGAR FLOW SWITCH" THEN
       "MANUAL INTERLOCK DB"."SUGAR UNHEALTHY" := 0;
   END_IF;
END_REGION

REGION Network 10: ------------------------------------------ CONTINUE RESET-------------------------------------
END_REGION

REGION Network 11: SYRUP MFG PROCESS ERROR FOR CONTINUE
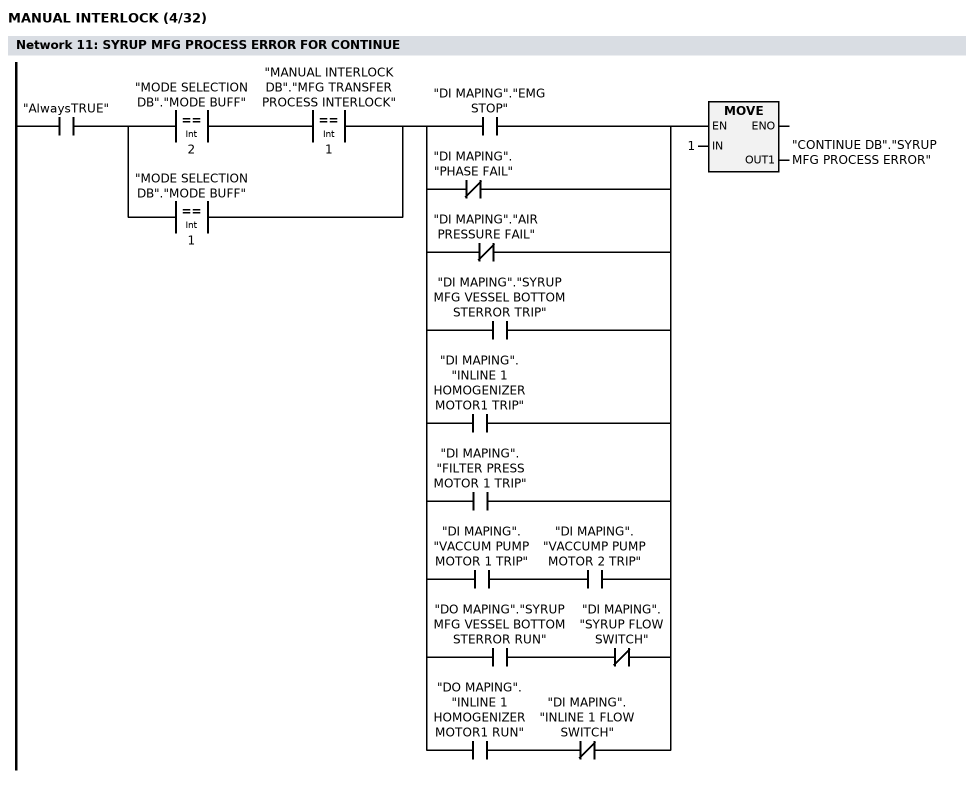
   RUNG wire#powerrail
      Contact( "AlwaysTRUE" )
      wire#w1
      { S7_Templates := "SrcType := Int" } EQ_Contact(in1 := "MODE SELECTION DB"."MODE BUFF", in2 := 2)
      { S7_Templates := "SrcType := Int" } EQ_Contact(in1 := "MANUAL INTERLOCK DB"."MFG TRANSFER PROCESS INTERLOCK", in2 := 1)
      wire#w2
      Contact( "DI MAPING"."EMG STOP" )
      wire#w3
      Move(in := 1, out1 => "CONTINUE DB"."SYRUP MFG PROCESS ERROR")
   END_RUNG
   RUNG wire#w1
      { S7_Templates := "SrcType := Int" } EQ_Contact(in1 := "MODE SELECTION DB"."MODE BUFF", in2 := 1)
   END_RUNG wire#w2
   RUNG wire#w2
      I_Contact( "DI MAPING"."PHASE FAIL" )
   END_RUNG wire#w3
   RUNG wire#w2
      I_Contact( "DI MAPING"."AIR PRESSURE FAIL" )
   END_RUNG wire#w3
   RUNG wire#w2
      Contact( "DI MAPING"."SYRUP MFG VESSEL BOTTOM STERROR TRIP" )
   END_RUNG wire#w3
   RUNG wire#w2
      Contact( "DI MAPING"."INLINE 1 HOMOGENIZER MOTOR1 TRIP" )
   END_RUNG wire#w3
   RUNG wire#w2
      Contact( "DI MAPING"."FILTER PRESS MOTOR 1 TRIP" )
   END_RUNG wire#w3
   RUNG wire#w2
      Contact( "DI MAPING"."VACCUM PUMP MOTOR 1 TRIP" )
      Contact( "DI MAPING"."VACCUMP PUMP MOTOR 2 TRIP" )
   END_RUNG wire#w3
   RUNG wire#w2
      Contact( "DO MAPING"."SYRUP MFG VESSEL BOTTOM STERROR RUN" )
      I_Contact( "DI MAPING"."SYRUP FLOW SWITCH" )
   END_RUNG wire#w3
   RUNG wire#w2
      Contact( "DO MAPING"."INLINE 1 HOMOGENIZER MOTOR1 RUN" )
      I_Contact( "DI MAPING"."INLINE 1 FLOW SWITCH" )
   END_RUNG wire#w3
   // the same network as SCL:
   IF "AlwaysTRUE" AND ((("MODE SELECTION DB"."MODE BUFF" = 2) AND ("MANUAL INTERLOCK DB"."MFG TRANSFER PROCESS INTERLOCK" = 1)) OR ("MODE SELECTION DB"."MODE BUFF" = 1)) AND ("DI MAPING"."EMG STOP" OR NOT "DI MAPING"."PHASE FAIL" OR NOT "DI MAPING"."AIR PRESSURE FAIL" OR "DI MAPING"."SYRUP MFG VESSEL BOTTOM STERROR TRIP" OR "DI MAPING"."INLINE 1 HOMOGENIZER MOTOR1 TRIP" OR "DI MAPING"."FILTER PRESS MOTOR 1 TRIP" OR ("DI MAPING"."VACCUM PUMP MOTOR 1 TRIP" AND "DI MAPING"."VACCUMP PUMP MOTOR 2 TRIP") OR ("DO MAPING"."SYRUP MFG VESSEL BOTTOM STERROR RUN" AND NOT "DI MAPING"."SYRUP FLOW SWITCH") OR ("DO MAPING"."INLINE 1 HOMOGENIZER MOTOR1 RUN" AND NOT "DI MAPING"."INLINE 1 FLOW SWITCH")) THEN
       "CONTINUE DB"."SYRUP MFG PROCESS ERROR" := 1;
   END_IF;
END_REGION

REGION Network 12: PREMIXING PROCESS ERROR FOR CONTINUE
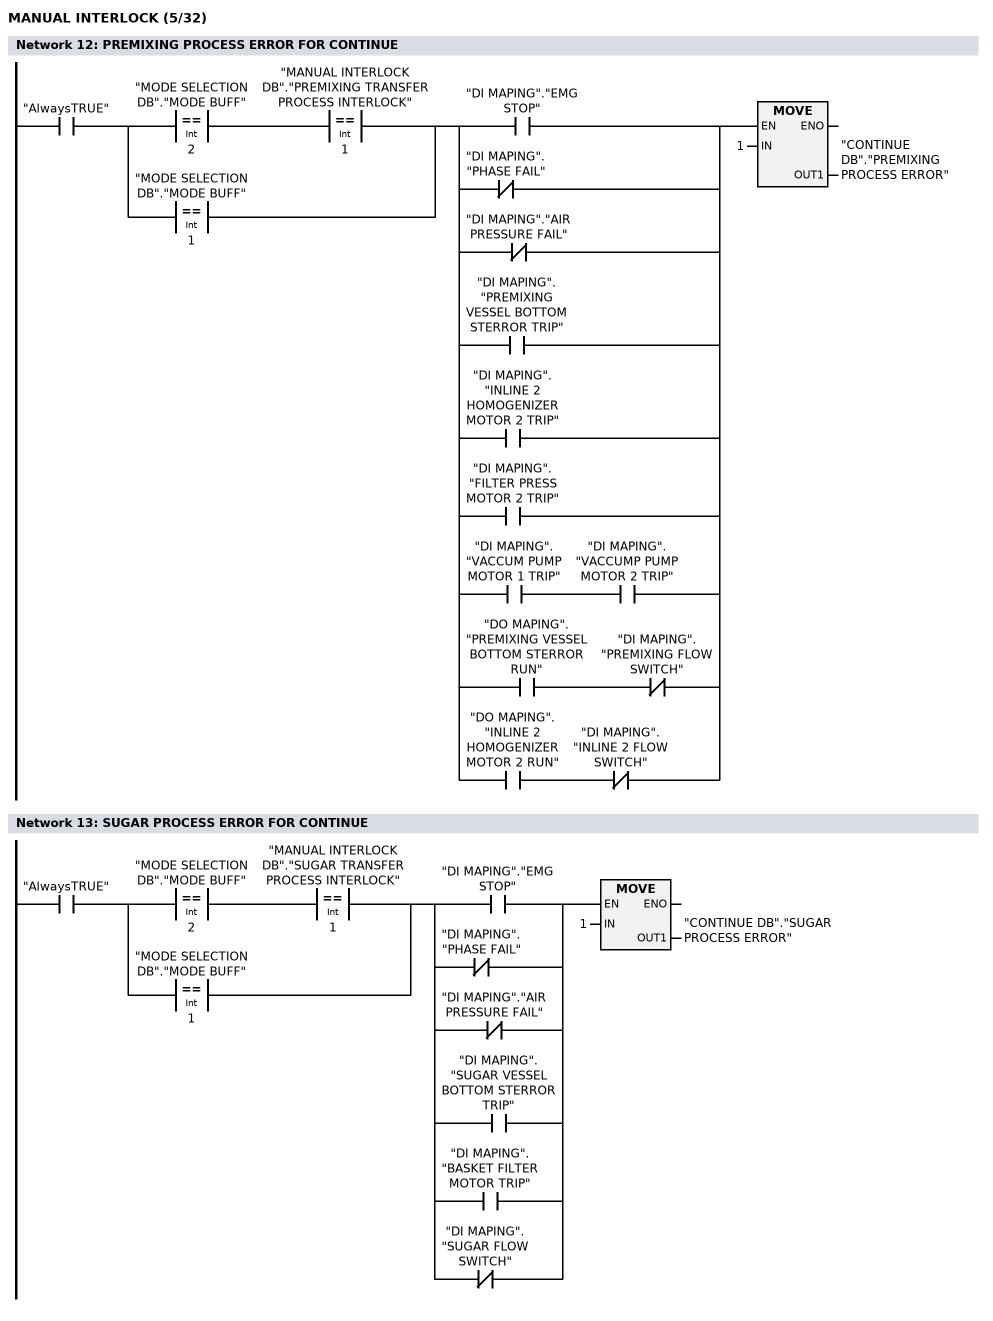
   RUNG wire#powerrail
      Contact( "AlwaysTRUE" )
      wire#w1
      { S7_Templates := "SrcType := Int" } EQ_Contact(in1 := "MODE SELECTION DB"."MODE BUFF", in2 := 2)
      { S7_Templates := "SrcType := Int" } EQ_Contact(in1 := "MANUAL INTERLOCK DB"."PREMIXING TRANSFER PROCESS INTERLOCK", in2 := 1)
      wire#w2
      Contact( "DI MAPING"."EMG STOP" )
      wire#w3
      Move(in := 1, out1 => "CONTINUE DB"."PREMIXING PROCESS ERROR")
   END_RUNG
   RUNG wire#w1
      { S7_Templates := "SrcType := Int" } EQ_Contact(in1 := "MODE SELECTION DB"."MODE BUFF", in2 := 1)
   END_RUNG wire#w2
   RUNG wire#w2
      I_Contact( "DI MAPING"."PHASE FAIL" )
   END_RUNG wire#w3
   RUNG wire#w2
      I_Contact( "DI MAPING"."AIR PRESSURE FAIL" )
   END_RUNG wire#w3
   RUNG wire#w2
      Contact( "DI MAPING"."PREMIXING VESSEL BOTTOM STERROR TRIP" )
   END_RUNG wire#w3
   RUNG wire#w2
      Contact( "DI MAPING"."INLINE 2 HOMOGENIZER MOTOR 2 TRIP" )
   END_RUNG wire#w3
   RUNG wire#w2
      Contact( "DI MAPING"."FILTER PRESS MOTOR 2 TRIP" )
   END_RUNG wire#w3
   RUNG wire#w2
      Contact( "DI MAPING"."VACCUM PUMP MOTOR 1 TRIP" )
      Contact( "DI MAPING"."VACCUMP PUMP MOTOR 2 TRIP" )
   END_RUNG wire#w3
   RUNG wire#w2
      Contact( "DO MAPING"."PREMIXING VESSEL BOTTOM STERROR RUN" )
      I_Contact( "DI MAPING"."PREMIXING FLOW SWITCH" )
   END_RUNG wire#w3
   RUNG wire#w2
      Contact( "DO MAPING"."INLINE 2 HOMOGENIZER MOTOR 2 RUN" )
      I_Contact( "DI MAPING"."INLINE 2 FLOW SWITCH" )
   END_RUNG wire#w3
   // the same network as SCL:
   IF "AlwaysTRUE" AND ((("MODE SELECTION DB"."MODE BUFF" = 2) AND ("MANUAL INTERLOCK DB"."PREMIXING TRANSFER PROCESS INTERLOCK" = 1)) OR ("MODE SELECTION DB"."MODE BUFF" = 1)) AND ("DI MAPING"."EMG STOP" OR NOT "DI MAPING"."PHASE FAIL" OR NOT "DI MAPING"."AIR PRESSURE FAIL" OR "DI MAPING"."PREMIXING VESSEL BOTTOM STERROR TRIP" OR "DI MAPING"."INLINE 2 HOMOGENIZER MOTOR 2 TRIP" OR "DI MAPING"."FILTER PRESS MOTOR 2 TRIP" OR ("DI MAPING"."VACCUM PUMP MOTOR 1 TRIP" AND "DI MAPING"."VACCUMP PUMP MOTOR 2 TRIP") OR ("DO MAPING"."PREMIXING VESSEL BOTTOM STERROR RUN" AND NOT "DI MAPING"."PREMIXING FLOW SWITCH") OR ("DO MAPING"."INLINE 2 HOMOGENIZER MOTOR 2 RUN" AND NOT "DI MAPING"."INLINE 2 FLOW SWITCH")) THEN
       "CONTINUE DB"."PREMIXING PROCESS ERROR" := 1;
   END_IF;
END_REGION

REGION Network 13: SUGAR PROCESS ERROR FOR CONTINUE
   RUNG wire#powerrail
      Contact( "AlwaysTRUE" )
      wire#w1
      { S7_Templates := "SrcType := Int" } EQ_Contact(in1 := "MODE SELECTION DB"."MODE BUFF", in2 := 2)
      { S7_Templates := "SrcType := Int" } EQ_Contact(in1 := "MANUAL INTERLOCK DB"."SUGAR TRANSFER PROCESS INTERLOCK", in2 := 1)
      wire#w2
      Contact( "DI MAPING"."EMG STOP" )
      wire#w3
      Move(in := 1, out1 => "CONTINUE DB"."SUGAR PROCESS ERROR")
   END_RUNG
   RUNG wire#w1
      { S7_Templates := "SrcType := Int" } EQ_Contact(in1 := "MODE SELECTION DB"."MODE BUFF", in2 := 1)
   END_RUNG wire#w2
   RUNG wire#w2
      I_Contact( "DI MAPING"."PHASE FAIL" )
   END_RUNG wire#w3
   RUNG wire#w2
      I_Contact( "DI MAPING"."AIR PRESSURE FAIL" )
   END_RUNG wire#w3
   RUNG wire#w2
      Contact( "DI MAPING"."SUGAR VESSEL BOTTOM STERROR TRIP" )
   END_RUNG wire#w3
   RUNG wire#w2
      Contact( "DI MAPING"."BASKET FILTER MOTOR TRIP" )
   END_RUNG wire#w3
   RUNG wire#w2
      I_Contact( "DI MAPING"."SUGAR FLOW SWITCH" )
   END_RUNG wire#w3
   // the same network as SCL:
   IF "AlwaysTRUE" AND ((("MODE SELECTION DB"."MODE BUFF" = 2) AND ("MANUAL INTERLOCK DB"."SUGAR TRANSFER PROCESS INTERLOCK" = 1)) OR ("MODE SELECTION DB"."MODE BUFF" = 1)) AND ("DI MAPING"."EMG STOP" OR NOT "DI MAPING"."PHASE FAIL" OR NOT "DI MAPING"."AIR PRESSURE FAIL" OR "DI MAPING"."SUGAR VESSEL BOTTOM STERROR TRIP" OR "DI MAPING"."BASKET FILTER MOTOR TRIP" OR NOT "DI MAPING"."SUGAR FLOW SWITCH") THEN
       "CONTINUE DB"."SUGAR PROCESS ERROR" := 1;
   END_IF;
END_REGION

REGION Network 15: CONTINUE PROCESS-SYRUP MFG
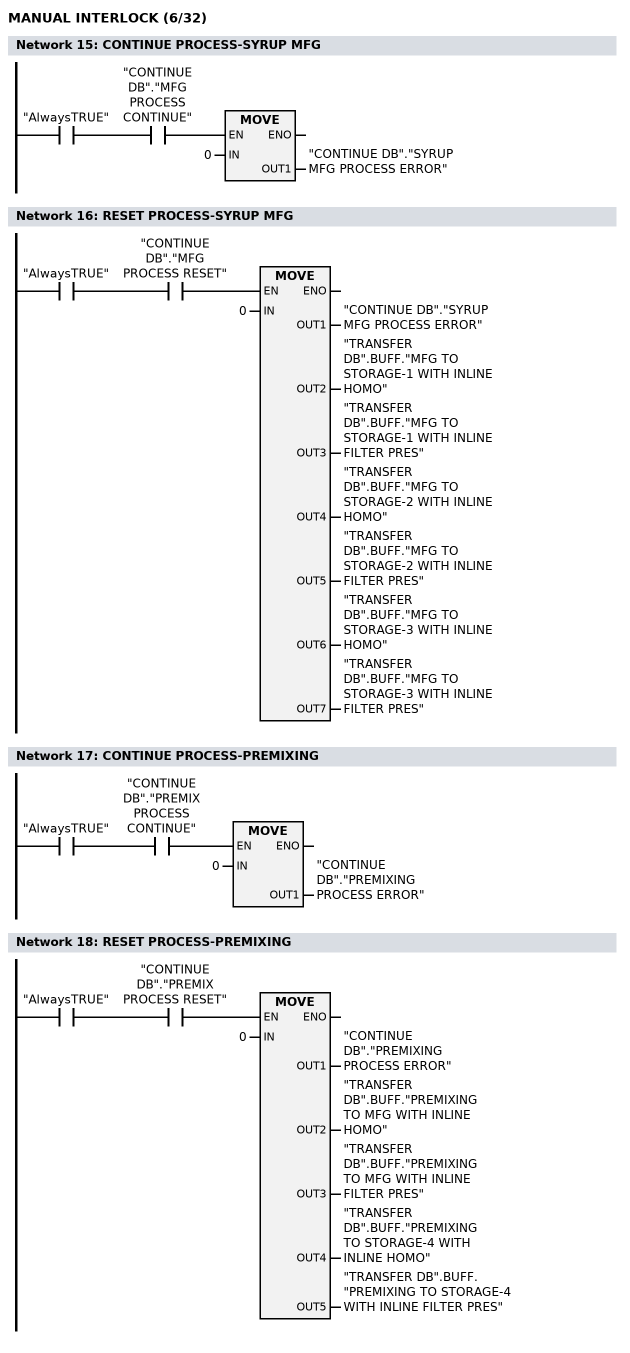
   RUNG wire#powerrail
      Contact( "AlwaysTRUE" )
      Contact( "CONTINUE DB"."MFG PROCESS CONTINUE" )
      Move(in := 0, out1 => "CONTINUE DB"."SYRUP MFG PROCESS ERROR")
   END_RUNG
   // the same network as SCL:
   IF "AlwaysTRUE" AND "CONTINUE DB"."MFG PROCESS CONTINUE" THEN
       "CONTINUE DB"."SYRUP MFG PROCESS ERROR" := 0;
   END_IF;
END_REGION

REGION Network 16: RESET PROCESS-SYRUP MFG
   RUNG wire#powerrail
      Contact( "AlwaysTRUE" )
      Contact( "CONTINUE DB"."MFG PROCESS RESET" )
      Move(in := 0, out1 => "CONTINUE DB"."SYRUP MFG PROCESS ERROR", out2 => "TRANSFER DB".BUFF."MFG TO STORAGE-1 WITH INLINE HOMO", out3 => "TRANSFER DB".BUFF."MFG TO STORAGE-1 WITH INLINE FILTER PRES", out4 => "TRANSFER DB".BUFF."MFG TO STORAGE-2 WITH INLINE HOMO", out5 => "TRANSFER DB".BUFF."MFG TO STORAGE-2 WITH INLINE FILTER PRES", out6 => "TRANSFER DB".BUFF."MFG TO STORAGE-3 WITH INLINE HOMO", out7 => "TRANSFER DB".BUFF."MFG TO STORAGE-3 WITH INLINE FILTER PRES")
   END_RUNG
   // the same network as SCL:
   IF "AlwaysTRUE" AND "CONTINUE DB"."MFG PROCESS RESET" THEN
       "CONTINUE DB"."SYRUP MFG PROCESS ERROR" := 0;
       "TRANSFER DB".BUFF."MFG TO STORAGE-1 WITH INLINE HOMO" := 0;
       "TRANSFER DB".BUFF."MFG TO STORAGE-1 WITH INLINE FILTER PRES" := 0;
       "TRANSFER DB".BUFF."MFG TO STORAGE-2 WITH INLINE HOMO" := 0;
       "TRANSFER DB".BUFF."MFG TO STORAGE-2 WITH INLINE FILTER PRES" := 0;
       "TRANSFER DB".BUFF."MFG TO STORAGE-3 WITH INLINE HOMO" := 0;
       "TRANSFER DB".BUFF."MFG TO STORAGE-3 WITH INLINE FILTER PRES" := 0;
   END_IF;
END_REGION

REGION Network 17: CONTINUE PROCESS-PREMIXING
   RUNG wire#powerrail
      Contact( "AlwaysTRUE" )
      Contact( "CONTINUE DB"."PREMIX PROCESS CONTINUE" )
      Move(in := 0, out1 => "CONTINUE DB"."PREMIXING PROCESS ERROR")
   END_RUNG
   // the same network as SCL:
   IF "AlwaysTRUE" AND "CONTINUE DB"."PREMIX PROCESS CONTINUE" THEN
       "CONTINUE DB"."PREMIXING PROCESS ERROR" := 0;
   END_IF;
END_REGION

REGION Network 18: RESET PROCESS-PREMIXING
   RUNG wire#powerrail
      Contact( "AlwaysTRUE" )
      Contact( "CONTINUE DB"."PREMIX PROCESS RESET" )
      Move(in := 0, out1 => "CONTINUE DB"."PREMIXING PROCESS ERROR", out2 => "TRANSFER DB".BUFF."PREMIXING TO MFG WITH INLINE HOMO", out3 => "TRANSFER DB".BUFF."PREMIXING TO MFG WITH INLINE FILTER PRES", out4 => "TRANSFER DB".BUFF."PREMIXING TO STORAGE-4 WITH INLINE HOMO", out5 => "TRANSFER DB".BUFF."PREMIXING TO STORAGE-4 WITH INLINE FILTER PRES")
   END_RUNG
   // the same network as SCL:
   IF "AlwaysTRUE" AND "CONTINUE DB"."PREMIX PROCESS RESET" THEN
       "CONTINUE DB"."PREMIXING PROCESS ERROR" := 0;
       "TRANSFER DB".BUFF."PREMIXING TO MFG WITH INLINE HOMO" := 0;
       "TRANSFER DB".BUFF."PREMIXING TO MFG WITH INLINE FILTER PRES" := 0;
       "TRANSFER DB".BUFF."PREMIXING TO STORAGE-4 WITH INLINE HOMO" := 0;
       "TRANSFER DB".BUFF."PREMIXING TO STORAGE-4 WITH INLINE FILTER PRES" := 0;
   END_IF;
END_REGION

REGION Network 19: CONTINUE PROCESS-SUGAR
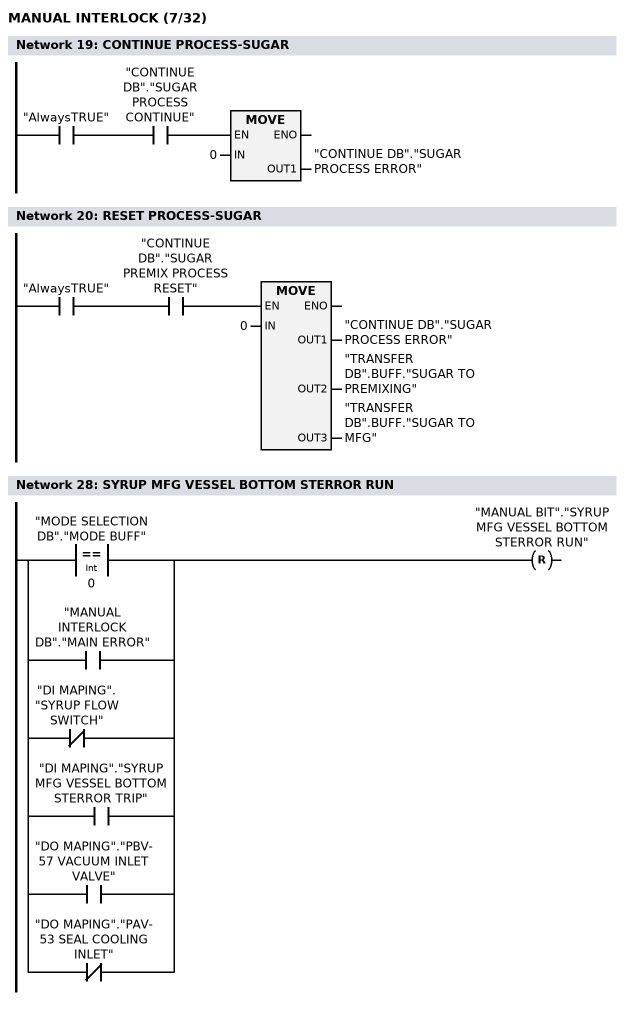
   RUNG wire#powerrail
      Contact( "AlwaysTRUE" )
      Contact( "CONTINUE DB"."SUGAR PROCESS CONTINUE" )
      Move(in := 0, out1 => "CONTINUE DB"."SUGAR PROCESS ERROR")
   END_RUNG
   // the same network as SCL:
   IF "AlwaysTRUE" AND "CONTINUE DB"."SUGAR PROCESS CONTINUE" THEN
       "CONTINUE DB"."SUGAR PROCESS ERROR" := 0;
   END_IF;
END_REGION

REGION Network 20: RESET PROCESS-SUGAR
   RUNG wire#powerrail
      Contact( "AlwaysTRUE" )
      Contact( "CONTINUE DB"."SUGAR PREMIX PROCESS RESET" )
      Move(in := 0, out1 => "CONTINUE DB"."SUGAR PROCESS ERROR", out2 => "TRANSFER DB".BUFF."SUGAR TO PREMIXING", out3 => "TRANSFER DB".BUFF."SUGAR TO MFG")
   END_RUNG
   // the same network as SCL:
   IF "AlwaysTRUE" AND "CONTINUE DB"."SUGAR PREMIX PROCESS RESET" THEN
       "CONTINUE DB"."SUGAR PROCESS ERROR" := 0;
       "TRANSFER DB".BUFF."SUGAR TO PREMIXING" := 0;
       "TRANSFER DB".BUFF."SUGAR TO MFG" := 0;
   END_IF;
END_REGION

REGION Network 22: ------------------------------TRANSFER PROCESS INTERLOCK---------------------------------------
END_REGION

REGION Network 23 (SCL): MFG TRANSFER PROCESS INTERLOCK
   IF 
       "TRANSFER DB".BUFF."MFG TO STORAGE-1 WITH INLINE HOMO" <> 0 OR
       "TRANSFER DB".BUFF."MFG TO STORAGE-1 WITH INLINE FILTER PRES" <> 0 OR
       "TRANSFER DB".BUFF."MFG TO STORAGE-2 WITH INLINE HOMO" <> 0 OR
       "TRANSFER DB".BUFF."MFG TO STORAGE-2 WITH INLINE FILTER PRES" <> 0 OR
       "TRANSFER DB".BUFF."MFG TO STORAGE-3 WITH INLINE HOMO" <> 0 OR
       "TRANSFER DB".BUFF."MFG TO STORAGE-3 WITH INLINE FILTER PRES" <> 0
   THEN
       "MANUAL INTERLOCK DB"."MFG TRANSFER PROCESS INTERLOCK" := 1;
   ELSIF "TRANSFER DB"."MFG VACCUM PUMP MOTOR-W 1 BIT"<>0
       OR "TRANSFER DB"."MFG VACCUMP PUMP MOTOR-S2 BIT"<>0
   THEN
       "MANUAL INTERLOCK DB"."MFG TRANSFER PROCESS INTERLOCK" := 2;
   ELSIF "RECIRCULATION DB".MFG.BUFF<>0
   THEN
       "MANUAL INTERLOCK DB"."MFG TRANSFER PROCESS INTERLOCK" := 3;
   ELSE
       "MANUAL INTERLOCK DB"."MFG TRANSFER PROCESS INTERLOCK" := 0;
   END_IF;
END_REGION

REGION Network 24 (SCL): PREMIXING TRANSFER PROCESS INTERLOCK
   IF
       "TRANSFER DB".BUFF."PREMIXING TO MFG WITH INLINE HOMO" <> 0 OR
       "TRANSFER DB".BUFF."PREMIXING TO MFG WITH INLINE FILTER PRES" <> 0 OR
       "TRANSFER DB".BUFF."PREMIXING TO STORAGE-4 WITH INLINE HOMO" <> 0 OR
       "TRANSFER DB".BUFF."PREMIXING TO STORAGE-4 WITH INLINE FILTER PRES" <> 0
   THEN
       "MANUAL INTERLOCK DB"."PREMIXING TRANSFER PROCESS INTERLOCK" := 1;
   ELSIF "TRANSFER DB"."PREMIXING VACCUM PUMP MOTOR-W 1 BIT"<>0 OR
       "TRANSFER DB"."PREMIXING VACCUMP PUMP MOTOR-S2 BIT"
   THEN
       "MANUAL INTERLOCK DB"."PREMIXING TRANSFER PROCESS INTERLOCK" := 2;
   ELSIF "RECIRCULATION DB".PREMIXING.BUFF<>0
   THEN
       "MANUAL INTERLOCK DB"."PREMIXING TRANSFER PROCESS INTERLOCK" := 3;
   ELSE
       "MANUAL INTERLOCK DB"."PREMIXING TRANSFER PROCESS INTERLOCK" := 0;
   END_IF;
END_REGION

REGION Network 25 (SCL): SUGAR TRANSFER PROCESS INTERLOCK
   IF "TRANSFER DB".BUFF."SUGAR TO PREMIXING" <>0 OR
       "TRANSFER DB".BUFF."SUGAR TO MFG"<>0
   THEN
       "MANUAL INTERLOCK DB"."SUGAR TRANSFER PROCESS INTERLOCK" := 1;
   ELSIF "DO MAPING"."PBV-30 VACUUM INLET VALVE" <>0
   THEN
       "MANUAL INTERLOCK DB"."SUGAR TRANSFER PROCESS INTERLOCK" := 2;
   ELSE
       "MANUAL INTERLOCK DB"."SUGAR TRANSFER PROCESS INTERLOCK" := 0;

   END_IF;
END_REGION

REGION Network 27: ------------------------------------------ MANUAL BIT RESET-------------------------------------
END_REGION

REGION Network 28: SYRUP MFG VESSEL BOTTOM STERROR RUN
   RUNG wire#powerrail
      { S7_Templates := "SrcType := Int" } EQ_Contact(in1 := "MODE SELECTION DB"."MODE BUFF", in2 := 0)
      wire#w1
      R_Coil( "MANUAL BIT"."SYRUP MFG VESSEL BOTTOM STERROR RUN" )
   END_RUNG
   RUNG wire#powerrail
      Contact( "MANUAL INTERLOCK DB"."MAIN ERROR" )
   END_RUNG wire#w1
   RUNG wire#powerrail
      I_Contact( "DI MAPING"."SYRUP FLOW SWITCH" )
   END_RUNG wire#w1
   RUNG wire#powerrail
      Contact( "DI MAPING"."SYRUP MFG VESSEL BOTTOM STERROR TRIP" )
   END_RUNG wire#w1
   RUNG wire#powerrail
      Contact( "DO MAPING"."PBV-57 VACUUM INLET VALVE" )
   END_RUNG wire#w1
   RUNG wire#powerrail
      I_Contact( "DO MAPING"."PAV-53 SEAL COOLING INLET" )
   END_RUNG wire#w1
   // the same network as SCL:
   IF ("MODE SELECTION DB"."MODE BUFF" = 0) OR "MANUAL INTERLOCK DB"."MAIN ERROR" OR NOT "DI MAPING"."SYRUP FLOW SWITCH" OR "DI MAPING"."SYRUP MFG VESSEL BOTTOM STERROR TRIP" OR "DO MAPING"."PBV-57 VACUUM INLET VALVE" OR NOT "DO MAPING"."PAV-53 SEAL COOLING INLET" THEN
       "MANUAL BIT"."SYRUP MFG VESSEL BOTTOM STERROR RUN" := FALSE;
   END_IF;
END_REGION

REGION Network 29: PREMIXING VESSEL BOTTOM STERROR RUN
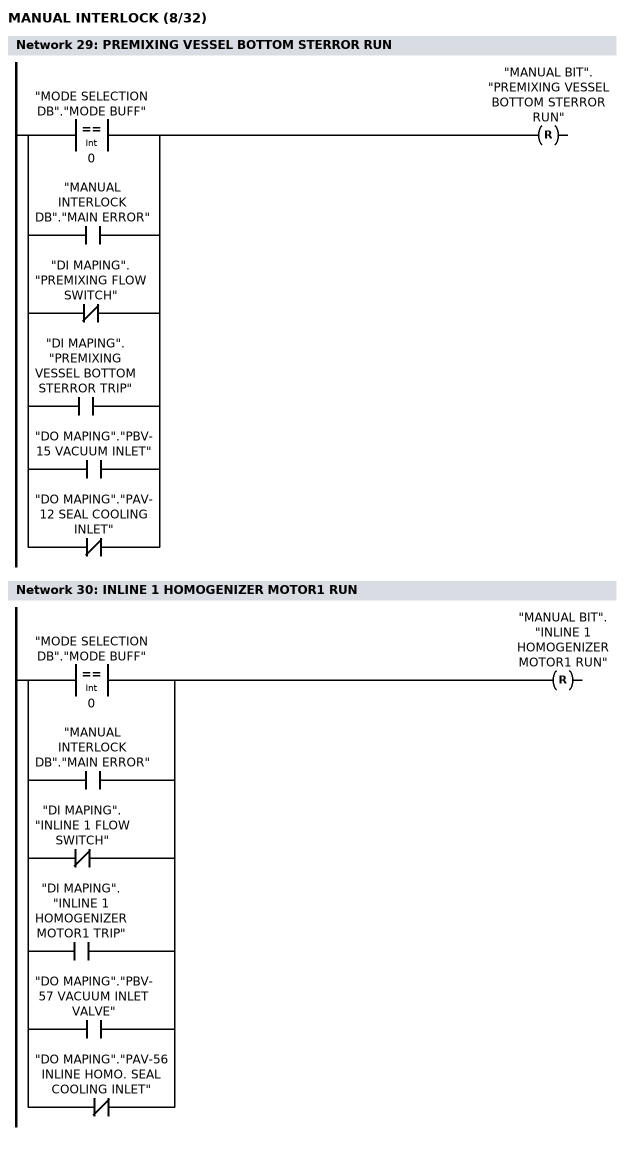
   RUNG wire#powerrail
      { S7_Templates := "SrcType := Int" } EQ_Contact(in1 := "MODE SELECTION DB"."MODE BUFF", in2 := 0)
      wire#w1
      R_Coil( "MANUAL BIT"."PREMIXING VESSEL BOTTOM STERROR RUN" )
   END_RUNG
   RUNG wire#powerrail
      Contact( "MANUAL INTERLOCK DB"."MAIN ERROR" )
   END_RUNG wire#w1
   RUNG wire#powerrail
      I_Contact( "DI MAPING"."PREMIXING FLOW SWITCH" )
   END_RUNG wire#w1
   RUNG wire#powerrail
      Contact( "DI MAPING"."PREMIXING VESSEL BOTTOM STERROR TRIP" )
   END_RUNG wire#w1
   RUNG wire#powerrail
      Contact( "DO MAPING"."PBV-15 VACUUM INLET" )
   END_RUNG wire#w1
   RUNG wire#powerrail
      I_Contact( "DO MAPING"."PAV-12 SEAL COOLING INLET" )
   END_RUNG wire#w1
   // the same network as SCL:
   IF ("MODE SELECTION DB"."MODE BUFF" = 0) OR "MANUAL INTERLOCK DB"."MAIN ERROR" OR NOT "DI MAPING"."PREMIXING FLOW SWITCH" OR "DI MAPING"."PREMIXING VESSEL BOTTOM STERROR TRIP" OR "DO MAPING"."PBV-15 VACUUM INLET" OR NOT "DO MAPING"."PAV-12 SEAL COOLING INLET" THEN
       "MANUAL BIT"."PREMIXING VESSEL BOTTOM STERROR RUN" := FALSE;
   END_IF;
END_REGION

REGION Network 30: INLINE 1 HOMOGENIZER MOTOR1 RUN
   RUNG wire#powerrail
      { S7_Templates := "SrcType := Int" } EQ_Contact(in1 := "MODE SELECTION DB"."MODE BUFF", in2 := 0)
      wire#w1
      R_Coil( "MANUAL BIT"."INLINE 1 HOMOGENIZER MOTOR1 RUN" )
   END_RUNG
   RUNG wire#powerrail
      Contact( "MANUAL INTERLOCK DB"."MAIN ERROR" )
   END_RUNG wire#w1
   RUNG wire#powerrail
      I_Contact( "DI MAPING"."INLINE 1 FLOW SWITCH" )
   END_RUNG wire#w1
   RUNG wire#powerrail
      Contact( "DI MAPING"."INLINE 1 HOMOGENIZER MOTOR1 TRIP" )
   END_RUNG wire#w1
   RUNG wire#powerrail
      Contact( "DO MAPING"."PBV-57 VACUUM INLET VALVE" )
   END_RUNG wire#w1
   RUNG wire#powerrail
      I_Contact( "DO MAPING"."PAV-56 INLINE HOMO. SEAL COOLING INLET" )
   END_RUNG wire#w1
   // the same network as SCL:
   IF ("MODE SELECTION DB"."MODE BUFF" = 0) OR "MANUAL INTERLOCK DB"."MAIN ERROR" OR NOT "DI MAPING"."INLINE 1 FLOW SWITCH" OR "DI MAPING"."INLINE 1 HOMOGENIZER MOTOR1 TRIP" OR "DO MAPING"."PBV-57 VACUUM INLET VALVE" OR NOT "DO MAPING"."PAV-56 INLINE HOMO. SEAL COOLING INLET" THEN
       "MANUAL BIT"."INLINE 1 HOMOGENIZER MOTOR1 RUN" := FALSE;
   END_IF;
END_REGION

REGION Network 31: INLINE 2 HOMOGENIZER MOTOR 2 RUN
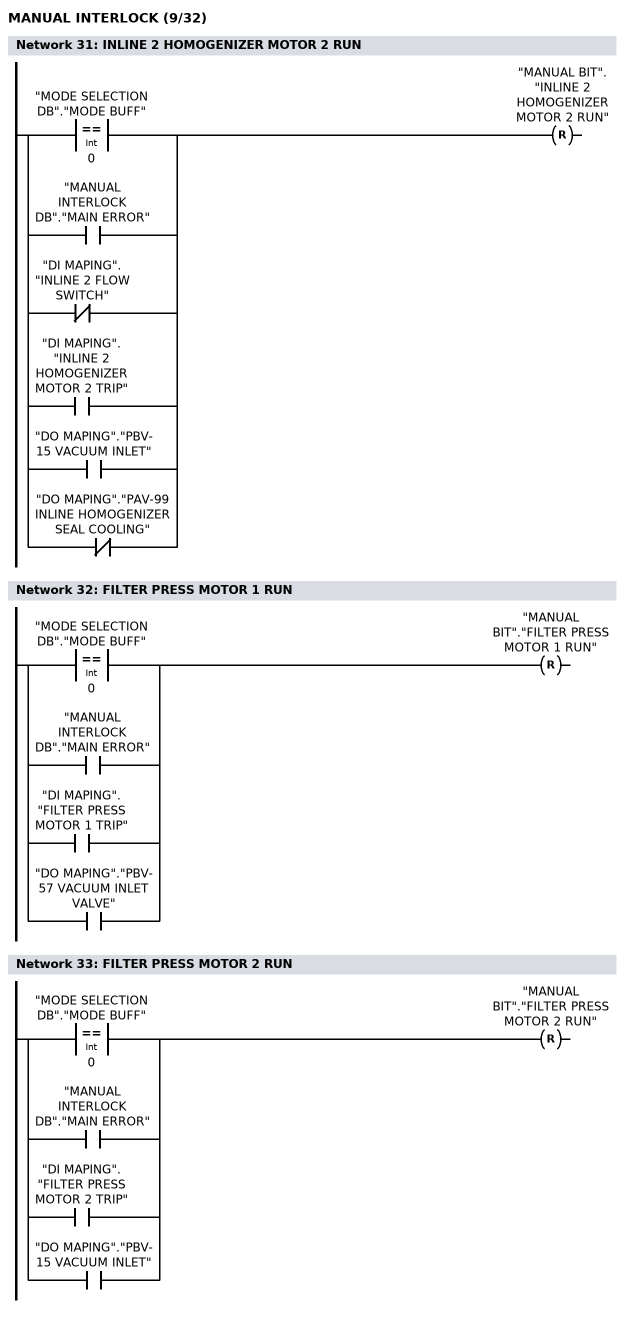
   RUNG wire#powerrail
      { S7_Templates := "SrcType := Int" } EQ_Contact(in1 := "MODE SELECTION DB"."MODE BUFF", in2 := 0)
      wire#w1
      R_Coil( "MANUAL BIT"."INLINE 2 HOMOGENIZER MOTOR 2 RUN" )
   END_RUNG
   RUNG wire#powerrail
      Contact( "MANUAL INTERLOCK DB"."MAIN ERROR" )
   END_RUNG wire#w1
   RUNG wire#powerrail
      I_Contact( "DI MAPING"."INLINE 2 FLOW SWITCH" )
   END_RUNG wire#w1
   RUNG wire#powerrail
      Contact( "DI MAPING"."INLINE 2 HOMOGENIZER MOTOR 2 TRIP" )
   END_RUNG wire#w1
   RUNG wire#powerrail
      Contact( "DO MAPING"."PBV-15 VACUUM INLET" )
   END_RUNG wire#w1
   RUNG wire#powerrail
      I_Contact( "DO MAPING"."PAV-99 INLINE HOMOGENIZER SEAL COOLING" )
   END_RUNG wire#w1
   // the same network as SCL:
   IF ("MODE SELECTION DB"."MODE BUFF" = 0) OR "MANUAL INTERLOCK DB"."MAIN ERROR" OR NOT "DI MAPING"."INLINE 2 FLOW SWITCH" OR "DI MAPING"."INLINE 2 HOMOGENIZER MOTOR 2 TRIP" OR "DO MAPING"."PBV-15 VACUUM INLET" OR NOT "DO MAPING"."PAV-99 INLINE HOMOGENIZER SEAL COOLING" THEN
       "MANUAL BIT"."INLINE 2 HOMOGENIZER MOTOR 2 RUN" := FALSE;
   END_IF;
END_REGION

REGION Network 32: FILTER PRESS MOTOR 1 RUN
   RUNG wire#powerrail
      { S7_Templates := "SrcType := Int" } EQ_Contact(in1 := "MODE SELECTION DB"."MODE BUFF", in2 := 0)
      wire#w1
      R_Coil( "MANUAL BIT"."FILTER PRESS MOTOR 1 RUN" )
   END_RUNG
   RUNG wire#powerrail
      Contact( "MANUAL INTERLOCK DB"."MAIN ERROR" )
   END_RUNG wire#w1
   RUNG wire#powerrail
      Contact( "DI MAPING"."FILTER PRESS MOTOR 1 TRIP" )
   END_RUNG wire#w1
   RUNG wire#powerrail
      Contact( "DO MAPING"."PBV-57 VACUUM INLET VALVE" )
   END_RUNG wire#w1
   // the same network as SCL:
   IF ("MODE SELECTION DB"."MODE BUFF" = 0) OR "MANUAL INTERLOCK DB"."MAIN ERROR" OR "DI MAPING"."FILTER PRESS MOTOR 1 TRIP" OR "DO MAPING"."PBV-57 VACUUM INLET VALVE" THEN
       "MANUAL BIT"."FILTER PRESS MOTOR 1 RUN" := FALSE;
   END_IF;
END_REGION

REGION Network 33: FILTER PRESS MOTOR 2 RUN
   RUNG wire#powerrail
      { S7_Templates := "SrcType := Int" } EQ_Contact(in1 := "MODE SELECTION DB"."MODE BUFF", in2 := 0)
      wire#w1
      R_Coil( "MANUAL BIT"."FILTER PRESS MOTOR 2 RUN" )
   END_RUNG
   RUNG wire#powerrail
      Contact( "MANUAL INTERLOCK DB"."MAIN ERROR" )
   END_RUNG wire#w1
   RUNG wire#powerrail
      Contact( "DI MAPING"."FILTER PRESS MOTOR 2 TRIP" )
   END_RUNG wire#w1
   RUNG wire#powerrail
      Contact( "DO MAPING"."PBV-15 VACUUM INLET" )
   END_RUNG wire#w1
   // the same network as SCL:
   IF ("MODE SELECTION DB"."MODE BUFF" = 0) OR "MANUAL INTERLOCK DB"."MAIN ERROR" OR "DI MAPING"."FILTER PRESS MOTOR 2 TRIP" OR "DO MAPING"."PBV-15 VACUUM INLET" THEN
       "MANUAL BIT"."FILTER PRESS MOTOR 2 RUN" := FALSE;
   END_IF;
END_REGION

REGION Network 34: VACCUM PUMP MOTOR 1 RUN
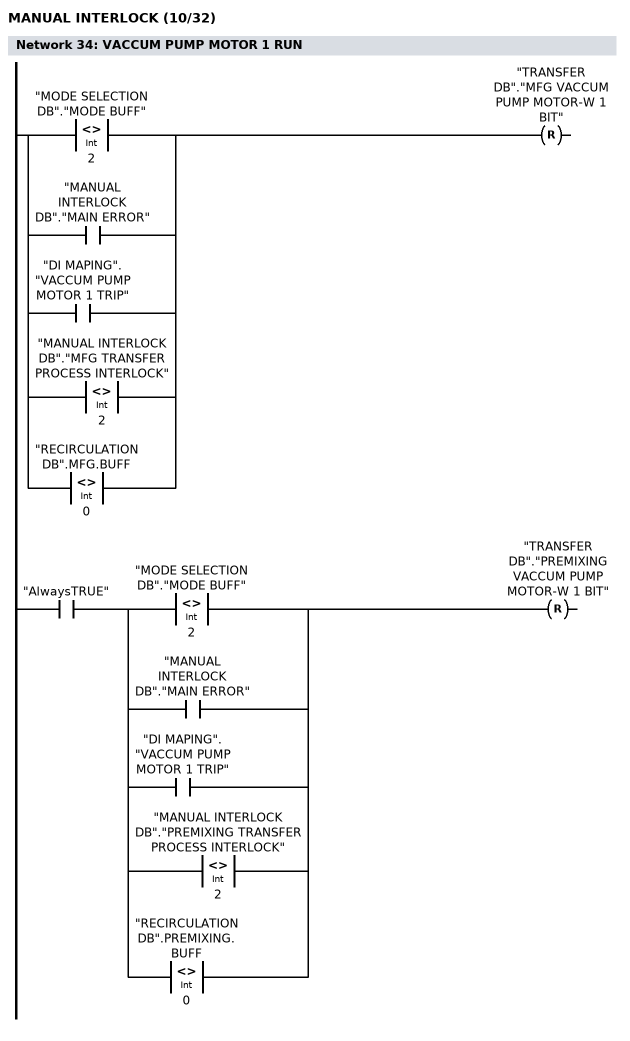
   RUNG wire#powerrail
      { S7_Templates := "SrcType := Int" } NE_Contact(in1 := "MODE SELECTION DB"."MODE BUFF", in2 := 2)
      wire#w1
      R_Coil( "TRANSFER DB"."MFG VACCUM PUMP MOTOR-W 1 BIT" )
   END_RUNG
   RUNG wire#powerrail
      Contact( "MANUAL INTERLOCK DB"."MAIN ERROR" )
   END_RUNG wire#w1
   RUNG wire#powerrail
      Contact( "DI MAPING"."VACCUM PUMP MOTOR 1 TRIP" )
   END_RUNG wire#w1
   RUNG wire#powerrail
      { S7_Templates := "SrcType := Int" } NE_Contact(in1 := "MANUAL INTERLOCK DB"."MFG TRANSFER PROCESS INTERLOCK", in2 := 2)
   END_RUNG wire#w1
   RUNG wire#powerrail
      { S7_Templates := "SrcType := Int" } NE_Contact(in1 := "RECIRCULATION DB".MFG.BUFF, in2 := 0)
   END_RUNG wire#w1
   RUNG wire#powerrail
      Contact( "AlwaysTRUE" )
      wire#w2
      { S7_Templates := "SrcType := Int" } NE_Contact(in1 := "MODE SELECTION DB"."MODE BUFF", in2 := 2)
      wire#w3
      R_Coil( "TRANSFER DB"."PREMIXING VACCUM PUMP MOTOR-W 1 BIT" )
   END_RUNG
   RUNG wire#w2
      Contact( "MANUAL INTERLOCK DB"."MAIN ERROR" )
   END_RUNG wire#w3
   RUNG wire#w2
      Contact( "DI MAPING"."VACCUM PUMP MOTOR 1 TRIP" )
   END_RUNG wire#w3
   RUNG wire#w2
      { S7_Templates := "SrcType := Int" } NE_Contact(in1 := "MANUAL INTERLOCK DB"."PREMIXING TRANSFER PROCESS INTERLOCK", in2 := 2)
   END_RUNG wire#w3
   RUNG wire#w2
      { S7_Templates := "SrcType := Int" } NE_Contact(in1 := "RECIRCULATION DB".PREMIXING.BUFF, in2 := 0)
   END_RUNG wire#w3
   // the same network as SCL:
   IF ("MODE SELECTION DB"."MODE BUFF" <> 2) OR "MANUAL INTERLOCK DB"."MAIN ERROR" OR "DI MAPING"."VACCUM PUMP MOTOR 1 TRIP" OR ("MANUAL INTERLOCK DB"."MFG TRANSFER PROCESS INTERLOCK" <> 2) OR ("RECIRCULATION DB".MFG.BUFF <> 0) THEN
       "TRANSFER DB"."MFG VACCUM PUMP MOTOR-W 1 BIT" := FALSE;
   END_IF;
   IF "AlwaysTRUE" AND (("MODE SELECTION DB"."MODE BUFF" <> 2) OR "MANUAL INTERLOCK DB"."MAIN ERROR" OR "DI MAPING"."VACCUM PUMP MOTOR 1 TRIP" OR ("MANUAL INTERLOCK DB"."PREMIXING TRANSFER PROCESS INTERLOCK" <> 2) OR ("RECIRCULATION DB".PREMIXING.BUFF <> 0)) THEN
       "TRANSFER DB"."PREMIXING VACCUM PUMP MOTOR-W 1 BIT" := FALSE;
   END_IF;
END_REGION

REGION Network 35: VACCUMP PUMP MOTOR 2 RUN
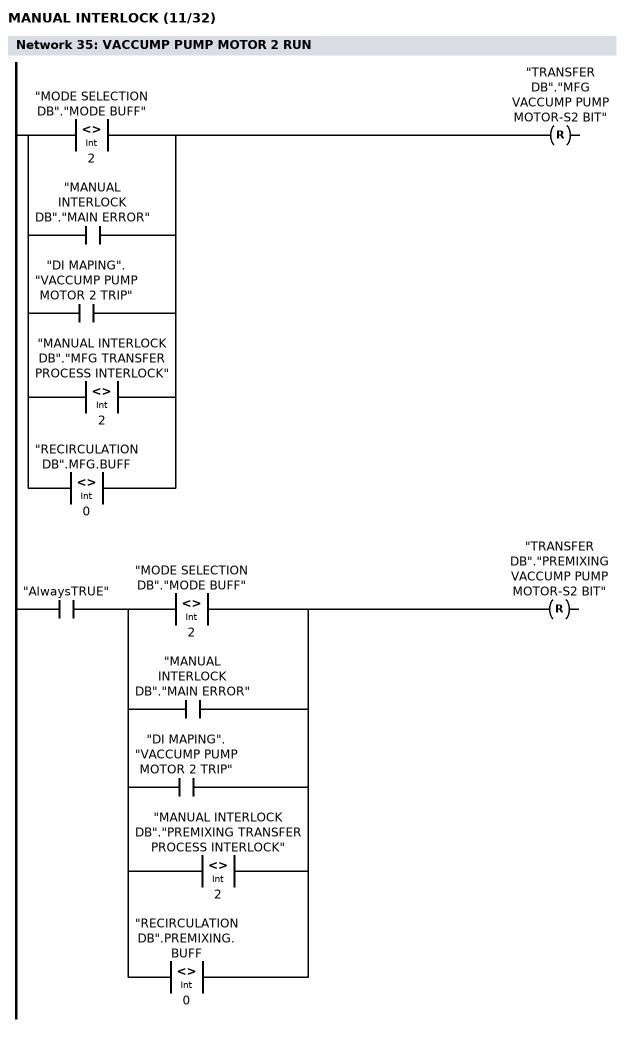
   RUNG wire#powerrail
      { S7_Templates := "SrcType := Int" } NE_Contact(in1 := "MODE SELECTION DB"."MODE BUFF", in2 := 2)
      wire#w1
      R_Coil( "TRANSFER DB"."MFG VACCUMP PUMP MOTOR-S2 BIT" )
   END_RUNG
   RUNG wire#powerrail
      Contact( "MANUAL INTERLOCK DB"."MAIN ERROR" )
   END_RUNG wire#w1
   RUNG wire#powerrail
      Contact( "DI MAPING"."VACCUMP PUMP MOTOR 2 TRIP" )
   END_RUNG wire#w1
   RUNG wire#powerrail
      { S7_Templates := "SrcType := Int" } NE_Contact(in1 := "MANUAL INTERLOCK DB"."MFG TRANSFER PROCESS INTERLOCK", in2 := 2)
   END_RUNG wire#w1
   RUNG wire#powerrail
      { S7_Templates := "SrcType := Int" } NE_Contact(in1 := "RECIRCULATION DB".MFG.BUFF, in2 := 0)
   END_RUNG wire#w1
   RUNG wire#powerrail
      Contact( "AlwaysTRUE" )
      wire#w2
      { S7_Templates := "SrcType := Int" } NE_Contact(in1 := "MODE SELECTION DB"."MODE BUFF", in2 := 2)
      wire#w3
      R_Coil( "TRANSFER DB"."PREMIXING VACCUMP PUMP MOTOR-S2 BIT" )
   END_RUNG
   RUNG wire#w2
      Contact( "MANUAL INTERLOCK DB"."MAIN ERROR" )
   END_RUNG wire#w3
   RUNG wire#w2
      Contact( "DI MAPING"."VACCUMP PUMP MOTOR 2 TRIP" )
   END_RUNG wire#w3
   RUNG wire#w2
      { S7_Templates := "SrcType := Int" } NE_Contact(in1 := "MANUAL INTERLOCK DB"."PREMIXING TRANSFER PROCESS INTERLOCK", in2 := 2)
   END_RUNG wire#w3
   RUNG wire#w2
      { S7_Templates := "SrcType := Int" } NE_Contact(in1 := "RECIRCULATION DB".PREMIXING.BUFF, in2 := 0)
   END_RUNG wire#w3
   // the same network as SCL:
   IF ("MODE SELECTION DB"."MODE BUFF" <> 2) OR "MANUAL INTERLOCK DB"."MAIN ERROR" OR "DI MAPING"."VACCUMP PUMP MOTOR 2 TRIP" OR ("MANUAL INTERLOCK DB"."MFG TRANSFER PROCESS INTERLOCK" <> 2) OR ("RECIRCULATION DB".MFG.BUFF <> 0) THEN
       "TRANSFER DB"."MFG VACCUMP PUMP MOTOR-S2 BIT" := FALSE;
   END_IF;
   IF "AlwaysTRUE" AND (("MODE SELECTION DB"."MODE BUFF" <> 2) OR "MANUAL INTERLOCK DB"."MAIN ERROR" OR "DI MAPING"."VACCUMP PUMP MOTOR 2 TRIP" OR ("MANUAL INTERLOCK DB"."PREMIXING TRANSFER PROCESS INTERLOCK" <> 2) OR ("RECIRCULATION DB".PREMIXING.BUFF <> 0)) THEN
       "TRANSFER DB"."PREMIXING VACCUMP PUMP MOTOR-S2 BIT" := FALSE;
   END_IF;
END_REGION

REGION Network 36: VACCUMP PUMP MOTOR 3 RUN
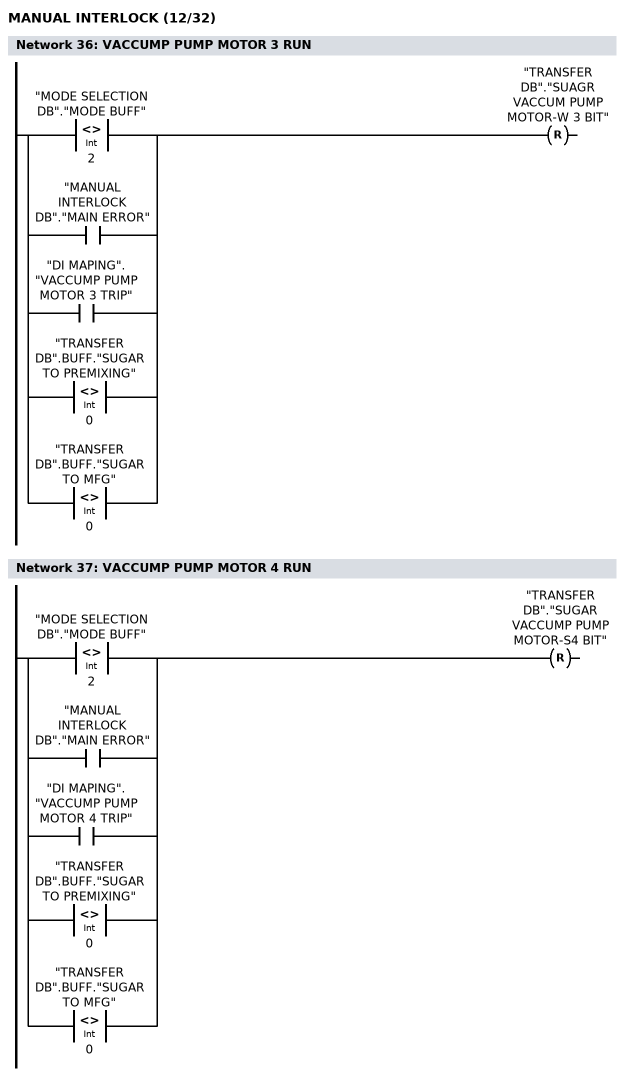
   RUNG wire#powerrail
      { S7_Templates := "SrcType := Int" } NE_Contact(in1 := "MODE SELECTION DB"."MODE BUFF", in2 := 2)
      wire#w1
      R_Coil( "TRANSFER DB"."SUAGR VACCUM PUMP MOTOR-W 3 BIT" )
   END_RUNG
   RUNG wire#powerrail
      Contact( "MANUAL INTERLOCK DB"."MAIN ERROR" )
   END_RUNG wire#w1
   RUNG wire#powerrail
      Contact( "DI MAPING"."VACCUMP PUMP MOTOR 3 TRIP" )
   END_RUNG wire#w1
   RUNG wire#powerrail
      { S7_Templates := "SrcType := Int" } NE_Contact(in1 := "TRANSFER DB".BUFF."SUGAR TO PREMIXING", in2 := 0)
   END_RUNG wire#w1
   RUNG wire#powerrail
      { S7_Templates := "SrcType := Int" } NE_Contact(in1 := "TRANSFER DB".BUFF."SUGAR TO MFG", in2 := 0)
   END_RUNG wire#w1
   // the same network as SCL:
   IF ("MODE SELECTION DB"."MODE BUFF" <> 2) OR "MANUAL INTERLOCK DB"."MAIN ERROR" OR "DI MAPING"."VACCUMP PUMP MOTOR 3 TRIP" OR ("TRANSFER DB".BUFF."SUGAR TO PREMIXING" <> 0) OR ("TRANSFER DB".BUFF."SUGAR TO MFG" <> 0) THEN
       "TRANSFER DB"."SUAGR VACCUM PUMP MOTOR-W 3 BIT" := FALSE;
   END_IF;
END_REGION

REGION Network 37: VACCUMP PUMP MOTOR 4 RUN
   RUNG wire#powerrail
      { S7_Templates := "SrcType := Int" } NE_Contact(in1 := "MODE SELECTION DB"."MODE BUFF", in2 := 2)
      wire#w1
      R_Coil( "TRANSFER DB"."SUGAR VACCUMP PUMP MOTOR-S4 BIT" )
   END_RUNG
   RUNG wire#powerrail
      Contact( "MANUAL INTERLOCK DB"."MAIN ERROR" )
   END_RUNG wire#w1
   RUNG wire#powerrail
      Contact( "DI MAPING"."VACCUMP PUMP MOTOR 4 TRIP" )
   END_RUNG wire#w1
   RUNG wire#powerrail
      { S7_Templates := "SrcType := Int" } NE_Contact(in1 := "TRANSFER DB".BUFF."SUGAR TO PREMIXING", in2 := 0)
   END_RUNG wire#w1
   RUNG wire#powerrail
      { S7_Templates := "SrcType := Int" } NE_Contact(in1 := "TRANSFER DB".BUFF."SUGAR TO MFG", in2 := 0)
   END_RUNG wire#w1
   // the same network as SCL:
   IF ("MODE SELECTION DB"."MODE BUFF" <> 2) OR "MANUAL INTERLOCK DB"."MAIN ERROR" OR "DI MAPING"."VACCUMP PUMP MOTOR 4 TRIP" OR ("TRANSFER DB".BUFF."SUGAR TO PREMIXING" <> 0) OR ("TRANSFER DB".BUFF."SUGAR TO MFG" <> 0) THEN
       "TRANSFER DB"."SUGAR VACCUMP PUMP MOTOR-S4 BIT" := FALSE;
   END_IF;
END_REGION

REGION Network 38: SUGAR VESSEL BOTTOM STERROR RUN
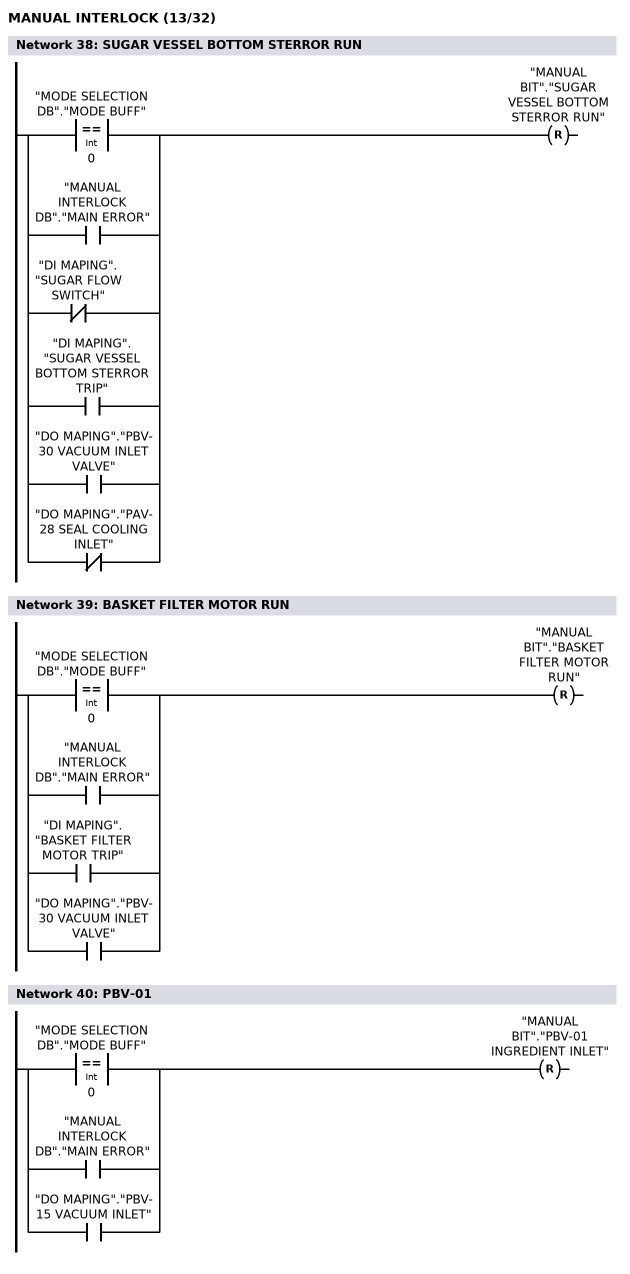
   RUNG wire#powerrail
      { S7_Templates := "SrcType := Int" } EQ_Contact(in1 := "MODE SELECTION DB"."MODE BUFF", in2 := 0)
      wire#w1
      R_Coil( "MANUAL BIT"."SUGAR VESSEL BOTTOM STERROR RUN" )
   END_RUNG
   RUNG wire#powerrail
      Contact( "MANUAL INTERLOCK DB"."MAIN ERROR" )
   END_RUNG wire#w1
   RUNG wire#powerrail
      I_Contact( "DI MAPING"."SUGAR FLOW SWITCH" )
   END_RUNG wire#w1
   RUNG wire#powerrail
      Contact( "DI MAPING"."SUGAR VESSEL BOTTOM STERROR TRIP" )
   END_RUNG wire#w1
   RUNG wire#powerrail
      Contact( "DO MAPING"."PBV-30 VACUUM INLET VALVE" )
   END_RUNG wire#w1
   RUNG wire#powerrail
      I_Contact( "DO MAPING"."PAV-28 SEAL COOLING INLET" )
   END_RUNG wire#w1
   // the same network as SCL:
   IF ("MODE SELECTION DB"."MODE BUFF" = 0) OR "MANUAL INTERLOCK DB"."MAIN ERROR" OR NOT "DI MAPING"."SUGAR FLOW SWITCH" OR "DI MAPING"."SUGAR VESSEL BOTTOM STERROR TRIP" OR "DO MAPING"."PBV-30 VACUUM INLET VALVE" OR NOT "DO MAPING"."PAV-28 SEAL COOLING INLET" THEN
       "MANUAL BIT"."SUGAR VESSEL BOTTOM STERROR RUN" := FALSE;
   END_IF;
END_REGION

REGION Network 39: BASKET FILTER MOTOR RUN
   RUNG wire#powerrail
      { S7_Templates := "SrcType := Int" } EQ_Contact(in1 := "MODE SELECTION DB"."MODE BUFF", in2 := 0)
      wire#w1
      R_Coil( "MANUAL BIT"."BASKET FILTER MOTOR RUN" )
   END_RUNG
   RUNG wire#powerrail
      Contact( "MANUAL INTERLOCK DB"."MAIN ERROR" )
   END_RUNG wire#w1
   RUNG wire#powerrail
      Contact( "DI MAPING"."BASKET FILTER MOTOR TRIP" )
   END_RUNG wire#w1
   RUNG wire#powerrail
      Contact( "DO MAPING"."PBV-30 VACUUM INLET VALVE" )
   END_RUNG wire#w1
   // the same network as SCL:
   IF ("MODE SELECTION DB"."MODE BUFF" = 0) OR "MANUAL INTERLOCK DB"."MAIN ERROR" OR "DI MAPING"."BASKET FILTER MOTOR TRIP" OR "DO MAPING"."PBV-30 VACUUM INLET VALVE" THEN
       "MANUAL BIT"."BASKET FILTER MOTOR RUN" := FALSE;
   END_IF;
END_REGION

REGION Network 40: PBV-01
   RUNG wire#powerrail
      { S7_Templates := "SrcType := Int" } EQ_Contact(in1 := "MODE SELECTION DB"."MODE BUFF", in2 := 0)
      wire#w1
      R_Coil( "MANUAL BIT"."PBV-01 INGREDIENT INLET" )
   END_RUNG
   RUNG wire#powerrail
      Contact( "MANUAL INTERLOCK DB"."MAIN ERROR" )
   END_RUNG wire#w1
   RUNG wire#powerrail
      Contact( "DO MAPING"."PBV-15 VACUUM INLET" )
   END_RUNG wire#w1
   // the same network as SCL:
   IF ("MODE SELECTION DB"."MODE BUFF" = 0) OR "MANUAL INTERLOCK DB"."MAIN ERROR" OR "DO MAPING"."PBV-15 VACUUM INLET" THEN
       "MANUAL BIT"."PBV-01 INGREDIENT INLET" := FALSE;
   END_IF;
END_REGION

REGION Network 41: PBV-02
